// TwinCAT 3 PLC project Tc3_1CNCPLCBase
// Title: CNC PLC Project
// Company: Beckhoff Automation GmbH & Co. KG
// ProjectVersion: 3.1.3035.30
// ProgramVersion: 3.1.4020.0
// libraries:
//   Tc2_CncHli, * (Beckhoff Automation GmbH)
//   Tc2_Drive, * (Beckhoff Automation GmbH)
//   Tc2_EtherCAT, * (Beckhoff Automation GmbH)
//   Tc2_IoFunctions, * (Beckhoff Automation GmbH)
//   Tc2_Standard, * (Beckhoff Automation GmbH)
//   Tc2_System, * (Beckhoff Automation GmbH)
//   Tc2_Utilities, * (Beckhoff Automation GmbH)
//   Tc3_Module, * (Beckhoff Automation GmbH)
// project tree:
//   CNC Beckhoff/1 Init/ HLI3_InitToolConfig.TcPOU, HLI3_Init.TcPOU, HLI3_SetAxisControlToPlc.TcPOU, HLI3_SetChannelControlToPlc.TcPOU, HLI3_UserInitialisation.TcPOU
//   CNC Beckhoff/2 OperationMode/ HLI3_AxisReset.TcPOU, HLI3_ChannelModeAuto.TcPOU, HLI3_ChannelModeManual.TcPOU, HLI3_ChannelModeMDI.TcPOU, HLI3_ChannelModeReference.TcPOU, HLI3_ChannelModeStandby.TcPOU, HLI3_ChannelReset.TcPOU, HLI3_ChannelResetRequest.TcPOU, HLI3_CNCChannel.TcPOU
//   CNC Beckhoff/2 OperationMode/ModeManual/ HLI3_LogicalAxisInManualMode.TcPOU, HLI3_ManualActivation.TcPOU, HLI3_ManualExecution.TcPOU, HLI3_ManualExecutionRapidMode.TcPOU, HLI3_ManualModeHandler.TcPOU, PRG_AnalogJoystick.TcPOU
//   CNC Beckhoff/3 Control/ FB_Diag.TcPOU, HLI3_ChannelSetBackwardMotion.TcPOU, HLI3_ChannelSetEmergencyStop.TcPOU, HLI3_ChannelSetFeedHold.TcPOU, HLI3_ChannelSetProgramBlockIgnore.TcPOU, HLI3_ChannelSetReducedFeed.TcPOU, HLI3_ChannelSetSingleBlock.TcPOU, HLI3_ChannelSetSuspendAxisOutput.TcPOU, HLI3_ClearReferencePosition.TcPOU, HLI3_GetActualAxisPos.TcPOU, HLI3_GetAxisReferenceState.TcPOU, HLI3_GetChannelActiveG.TcPOU, HLI3_GetChannelError.TcPOU, HLI3_GetChannelMessage.TcPOU, HLI3_GetChannelMode.TcPOU, HLI3_GetChannelState.TcPOU, HLI3_GetChannelStatusInfo.TcPOU, HLI3_GetEtherCATAxisInfo.TcPOU, HLI3_GetFeedholdState.TcPOU, HLI3_GetIpoState.TcPOU, HLI3_HandleSpindleTechno.TcPOU, HLI3_HandleSpindleTechnoGearchange.TcPOU, HLI3_SetAxisGantryOn.TcPOU, HLI3_SetAxisOverride.TcPOU, HLI3_SetAxisReferenceCam.TcPOU, HLI3_SetAxisReferencePosition.TcPOU, HLI3_SetAxisRelease.TcPOU, HLI3_SetAxisSpindleStopAtProgramEnd.TcPOU, HLI3_SetAxisTrackingOperation.TcPOU, HLI3_SetChannelOverride.TcPOU, HLI3_SetProbingSignal.TcPOU
//   CNC Beckhoff/4 MHT-Function/ HLI3_ChannelResetHFunctions.TcPOU, HLI3_ChannelResetMFunctions.TcPOU, HLI3_DoChannelHFunction.TcPOU, HLI3_DoChannelMFunction.TcPOU, HLI3_DoChannelTFunction.TcPOU, HLI3_FastMFunctionHandler.TcPOU, HLI3_FastMFunctionProvider.TcPOU, HLI3_QuitAxisMFunction.TcPOU, HLI3_QuitChannelMHTFunction.TcPOU, PRG_FastMFunctions.TcPOU
//   CNC Beckhoff/5 Variables/ FB_ReadCNCVariables.TcPOU, HLI3_GetVEChannelDIntValue.TcPOU, HLI3_GetVEChannelBooleanValue.TcPOU, HLI3_GetVEChannelLRealValue.TcPOU, HLI3_GetVEChannelStringValue.TcPOU, HLI3_LinkVEChannelStructure.TcPOU, HLI3_SetVEChannelDIntValue.TcPOU, HLI3_SetVEChannelBooleanValue.TcPOU, HLI3_SetVEChannelLRealValue.TcPOU, HLI3_SetVEChannelStringValue.TcPOU
//   CNC Beckhoff/6 BlockSearch/ HLI3_BlockSearch.TcPOU, ReadBlockCount.TcPOU, ReadBlockNumber.TcPOU, ReadBsAutoReturn.TcPOU, ReadBsBlockCount.TcPOU, ReadBsBlockNumber.TcPOU, ReadBsCoveredDistance.TcPOU, ReadBsDeviationMax.TcPOU, ReadBsPass.TcPOU, ReadBsType.TcPOU, WriteBsAutoReturn.TcPOU, WriteBsBlockCount.TcPOU, WriteBsBlockNumber.TcPOU, WriteBsCoveredDistance.TcPOU, WriteBsDeviationMax.TcPOU, WriteBsPass.TcPOU, WriteBsType.TcPOU
//   CNC Beckhoff/9 Mis/ ADSLOG.TcPOU, FB_WriteCNCZeroOffset.TcPOU, FB_WriteCNCZeroOffsetDefault.TcPOU, HLI3_CheckAxisValid.TcPOU, HLI3_CheckChannelValid.TcPOU, HLI3_CheckCNCAlive.TcPOU, HLI3_GetHliAxisIdx.TcPOU, HLI3_GetLogAxisId.TcPOU, HLI3_SetPLCAlive.TcPOU, HLI_HandleMessages.TcPOU, HLI_MoveSpindle.TcPOU, PB_10_CNC_Spindelkopplung.TcPOU, HLI3_ResetSpindle.TcPOU
//   CNC Beckhoff/Demo/ PRG_Demo.TcPOU, PRG_MachineStatusV2.TcPOU
//   CNC Beckhoff/Messages/ FB_ChannelError.TcPOU, FB_EventLog.TcPOU, FB_ExtSimpleEventLog.TcPOU, FB_SimpleEventLog.TcPOU
//   CNC Beckhoff/ PRG_AxesHandler.TcPOU, PRG_ChannelHandler.TcPOU, PRG_CNCVariablesViewer.TcPOU, PRG_ManualMode.TcPOU, PRG_ManualModeHMI.TcPOU, PRG_ShowMessages.TcPOU
//   CNC Beckhoff/Util/ Blinker.TcPOU, FB_CNCWriteParameter.TcPOU, FB_Uint_Udint.TcPOU, F_GRAYCODE_TO_UINT.TcPOU, HLI3_FindHliAxisIdx.TcPOU, HLI3_FindAxisNameAndChannel.TcPOU
//   Data types/CNC_DataTyps/ E_CNC_MM_Controller.TcDUT, E_HLI_MM_KEYDIRECTION.TcDUT, ST_BlockSearch.TcDUT, ST_ChannelSignals.TcDUT, ST_CNCAxis.TcDUT, ST_CncChannel.TcDUT, ST_CNCG159VG.TcDUT, ST_CncSystem.TcDUT, ST_CNC_TOOL_DATA_EXT.TcDUT, ST_ManualMode.TcDUT, ST_OpModes.TcDUT, ST_OpStates.TcDUT, ST_SyntaxCheck.TcDUT, ST_TechnoAttributeData.TcDUT, VEData.TcDUT
//   Data types/CNC_FastMFunction/ E_FastMFunctionState.TcDUT, ST_FastMFunctionBufferItem.TcDUT, ST_FastMFunctionData.TcDUT, ST_FastMFunctionItem.TcDUT
//   Data types/CNC_ManualMode/ E_CNC_ManualType.TcDUT, ST_ManualModeAxis.TcDUT, ST_ManualModeAxisKeys.TcDUT, ST_ManualModeAxisParameter.TcDUT, ST_ManualModeChannelParameter.TcDUT, ST_ManualModeControlElements.TcDUT, ST_ManualModeControlElementState.TcDUT, ST_ManualModeJoystickParameter.TcDUT, ST_ManualModeKeyHWUnit.TcDUT, ST_ManualModeParameter.TcDUT, ST_ManualModeState.TcDUT
//   Data types/CNC_VariablesViewer/ E_CNCVariablesType.TcDUT, E_VEVariablesType.TcDUT, ST_CNCVariablesViewer_Data.TcDUT
//   Data types/CNC_WriteParameter/ E_CNCParameterTypes.TcDUT, ST_CNCParameter.TcDUT
//   Data types/EtherCAT Diag/ E_EcCommState.TcDUT, ST_EcMasterDevState.TcDUT, ST_PortAddr.TcDUT, ST_SlaveState.TcDUT, ST_SlaveStateInfo.TcDUT, ST_SlaveStateInfoScanned.TcDUT, ST_TopologyData.TcDUT
//   Data types/EventLogger/ E_LogMethod.TcDUT, ST_EventData.TcDUT, ST_FileInfo.TcDUT
//   Data types/ E_HLI_MM_STATE.TcDUT, ST_Diagnose.TcDUT, ST_EtherCATAxisInfo.TcDUT, ST_EventData1.TcDUT, ST_EventDataAX5000_1.TcDUT, ST_MachineMode.TcDUT, ST_MViewStatus.TcDUT, ST_WKZDaten.TcDUT, ST_WPCounter.TcDUT
//   Data types/General SoE DTs/ ST_SoE_String.TcDUT, ST_SoE_StringEx.TcDUT
//   Data types/Magazin/ ST_Magazin.TcDUT
//   Data types/MaschinenDaten PlcStructure/ ST_HMIPDatMaschine.TcDUT, ST_HMIPDatProg.TcDUT, ST_HMI_Manual.TcDUT, ST_MachData.TcDUT, ST_PDatLineProgLine.TcDUT, ST_PDatLineProgValue.TcDUT
//   Data types/Recipe/ RecipeHeader_Struct.TcDUT, RecipeList_Struct.TcDUT
//   Data types/SERCOS/ E_SoE_AttribLen.TcDUT, E_SoE_CmdControl.TcDUT, E_SoE_CmdState.TcDUT, E_SoE_Type.TcDUT
//   / FAST.TcPOU, MAIN.TcPOU, PlcFastTask.TcTTO, Standard_Task.TcTTO
//   Global Variables/Examples/ Globale_EtherCATDiag.TcGVL, Global_BDE.TcGVL, Global_MachineView.TcGVL, Global_ManualPlcFunctions.TcGVL, Global_MaschinenDaten.TcGVL, Global_VE.TcGVL
//   Global Variables/ Global_CNC.TcGVL, Global_CNCVariablesViewer.TcGVL, Global_HMI.TcGVL, Global_ManualMode.TcGVL, Global_Messages.TcGVL, Variable_Configuration.TcGVL
//   Version/ Global_Version.TcGVL
// real-time tasks:
//   TASK Standard_Task: cycle T#10ms, priority 21, ADS port 350
//   TASK PlcFastTask: cycle T#1ms, priority 4, ADS port 351
// I/O:
//   DEVICE Gerät 3 (EtherCAT), AmsNetId 10.99.10.27.4.1
//     testachse [AX5103-0000-0203 EtherCAT Drive (SoE, 1 Ch.)] (disabled)
//     Drive 2 (AX5206-0000-0011) [AX5206-0000 EtherCAT Drive (SoE, 2 Ch.)]
// variable links:
//   CNC/Axes/Axis_2 <-> Device 3 (EtherCAT)/Drive 2 (AX5206-0000-0011)
//     Inputs/Drive status word <-> AT 1/Drive status word
//     Inputs/Following distance <-> AT 1/Following distance
//     Inputs/Position feedback value 1 (motor feedback) <-> AT 1/Position feedback value 1 (motor feedback)
//     Inputs/WcState <-> WcState/WcState
//     Outputs/Master control word <-> MDT 1/Master control word
//     Outputs/Position command value <-> MDT 1/Position command value
//   CNC/Axes/Axis_3 <-> Device 3 (EtherCAT)/Drive 2 (AX5206-0000-0011)
//     Inputs/Drive status word <-> AT 2/Drive status word
//     Inputs/Following distance <-> AT 2/Following distance
//     Inputs/Position feedback value 1 (motor feedback) <-> AT 2/Position feedback value 1 (motor feedback)
//     Inputs/WcState <-> WcState/WcState
//     Outputs/Master control word <-> MDT 2/Master control word
//     Outputs/Position command value <-> MDT 2/Position command value
//   Tc3_1CNCPLCBase/Tc3_1CNCPLCBase Instance <-> Device 3 (EtherCAT)/Drive 2 (AX5206-0000-0011)
//     Standard_Task Inputs/MAIN.DigitalIn <-> AT 1/Digital inputs, state
//     Standard_Task Outputs/MAIN.Trennscheibe <-> MDT 1/Digital outputs

CONFIGURATION Tc3_1CNCPLCBase
    RESOURCE PLC ON TwinCAT3
        TASK PlcFastTask(INTERVAL := T#1ms, PRIORITY := 4);
        TASK Standard_Task(INTERVAL := T#10ms, PRIORITY := 21);
        PROGRAM FAST WITH PlcFastTask : FAST;
        PROGRAM MAIN WITH Standard_Task : MAIN;
    END_RESOURCE
END_CONFIGURATION

// ---- Data types/CNC_DataTyps/E_CNC_MM_Controller.TcDUT
TYPE E_CNC_MM_Controller :
(
	HMI := 0,
	PANEL := 1,
	REMOTE := 2,
	CUSTOMER := 3
);
END_TYPE

// ---- Data types/CNC_DataTyps/E_HLI_MM_KEYDIRECTION.TcDUT
TYPE E_HLI_MM_KEYDIRECTION :
(
	KEY_DIR_NEGATIVE := -1,
	KEY_DIR_NOT_PRESSED := 0,
	KEY_DIR_POSITIVE := 1
);
END_TYPE

// ---- Data types/CNC_DataTyps/ST_BlockSearch.TcDUT
TYPE ST_BlockSearch :
STRUCT
	/// Block Search 
	Active: BOOL;
	/// Edge signal 
	bStartRead: BOOL;
	/// Edge signal 
	bStartWrite: BOOL;
	/// 0 - no block search
	///                                    3 - start position by block count
	///                                    4 - start position by block nr
	///                                    5 - start position BY individual mark 
	nType: UINT;
	fDistance: LREAL;
	bAutoReturn: BOOL;
	nDeviationMax: UDINT;
	nBlockNumber: DINT;
	nPass: DINT;
	nBlockCount: DINT;
END_STRUCT
END_TYPE

// ---- Data types/CNC_DataTyps/ST_ChannelSignals.TcDUT
TYPE ST_ChannelSignals :
STRUCT
	DoSingleBlock: BOOL;
	SingleBlock: BOOL;
	FeedHold: BOOL;
	Backward: BOOL;
	PrgBlockIgnore: BOOL;
	M01Stop: BOOL;
END_STRUCT
END_TYPE

// ---- Data types/CNC_DataTyps/ST_CNCAxis.TcDUT
TYPE ST_CNCAxis :
STRUCT
	nHliAxisIdx : INT := -1;
    stLogName	: STRING(HLI_ACHS_NAME_LAENGE);
END_STRUCT
END_TYPE

// ---- Data types/CNC_DataTyps/ST_CncChannel.TcDUT
TYPE ST_CncChannel :
STRUCT
	/// Operation Mode 
	Mode: ST_OpModes;
	/// Operation States 
	State: ST_OpStates;
	/// Selected Mode 
	ActMode: UDINT;
	/// Selected Mode as string 
	ActModeString: STRING;
	/// Selected State 
	ActState: UDINT;
	/// Selected State as string 
	ActStateString: STRING;
	/// Block Search : Act. Distance 
	ActDistance: LREAL;
	/// Block Search : Act. Block Count 
	ActBlockCount: UDINT;
	actM_r: STRING(5);
	actH_r: STRING(5);
	/// M-Functions 
	M: ARRAY[0..999] OF ST_TechnoAttributeData;
	/// H-Functions 
	H: ARRAY[0..999] OF ST_TechnoAttributeData;	
	/// Fehlerflag des Kanals 
	Error: BOOL;	
	/// Message from NC program to PLC 
	Message: STRING(HLI_MSG_CONTENT_STRL);
END_STRUCT
END_TYPE

// ---- Data types/CNC_DataTyps/ST_CNCG159VG.TcDUT
TYPE ST_CNCG159VG :
STRUCT
	sTarget: STRING(95);
	dValue: DINT;
END_STRUCT
END_TYPE

// ---- Data types/CNC_DataTyps/ST_CncSystem.TcDUT
TYPE ST_CncSystem :
STRUCT
	/// Initialization of HLI done 
	bHLIInit: BOOL;
	/// Initialization of user data done 
	bUserInitDone: BOOL;
	/// Error init HLI-Interfaces 
	bInitError: BOOL;
	/// ErrorId during init HLI-Interfaces 
	nInitErrorId: UDINT;
	Channel: ARRAY[0..HLI_SYS_CH_MAXIDX] OF ST_CncChannel;
    LogAxisNo : ARRAY[0..MAX_SYS_LOG_AXIS_INDEX] OF ST_CncAxis;	
END_STRUCT
END_TYPE

// ---- Data types/CNC_DataTyps/ST_CNC_TOOL_DATA_EXT.TcDUT
TYPE ST_CNC_TOOL_DATA_EXT :
STRUCT
	tool_desc: CNC_TOOL_DESC;
	tool_life: CNC_TOOL_LIFE_DATA;
	dist_max: LREAL;
	time_max: LREAL;
	/// 0.1 µm 
	laenge: DINT;
	/// 0.1 µm 
	laenge_delta: DINT;
	/// 0.1 µm 
	radius: DINT;
	/// 0.1 µm 
	radius_delta: DINT;
	/// position in tool holder 
	pos: DINT;
	/// 0.1 µm 
	tolerancePos: DINT;
	/// 0.1 µm 
	toleranceNeg: DINT;
END_STRUCT
END_TYPE

// ---- Data types/CNC_DataTyps/ST_ManualMode.TcDUT
TYPE ST_ManualMode :
STRUCT
	bKeyPos: BOOL;
	bKeyNeg: BOOL;
	bKeyRapid: BOOL;
	nLogAxisNumber: UINT;
	nInc: UDINT;
	nManualTyp: UINT;
	nSpeed: UINT;
	/// Handradauflösung in 0.1 um / Umdrehung 
	nHwResolution: UDINT;
END_STRUCT
END_TYPE

// ---- Data types/CNC_DataTyps/ST_OpModes.TcDUT
TYPE ST_OpModes :
STRUCT
	Standby: BOOL;
	Auto: BOOL;
	Manual: BOOL;
	MDI: BOOL;
	///Reference		: BOOL;  TC3HR
	Homing: BOOL;
END_STRUCT
END_TYPE

// ---- Data types/CNC_DataTyps/ST_OpStates.TcDUT
TYPE ST_OpStates :
STRUCT
	Selected: BOOL;
	Ready: BOOL;
	Start: BOOL;
	Stop: BOOL;
	Reset: BOOL;
END_STRUCT
END_TYPE

// ---- Data types/CNC_DataTyps/ST_SyntaxCheck.TcDUT
TYPE ST_SyntaxCheck :
STRUCT
	/// SyntaxCheck 
	nType: INT;
END_STRUCT
END_TYPE

// ---- Data types/CNC_DataTyps/ST_TechnoAttributeData.TcDUT
TYPE ST_TechnoAttributeData :
STRUCT
	bState_rw: BOOL;
	nFunctionNumber_r: UDINT;
	nTime_r: DINT;
	nBlockNumber_r: UDINT;
	nPrgLineNumber_r: UDINT;
	nArgument_r: DINT;
	bRes: BOOL;
END_STRUCT
END_TYPE

// ---- Data types/CNC_DataTyps/VEData.TcDUT
TYPE VEData :
STRUCT
	AHLI_UNS32_Data: ARRAY[0..HLI_EXT_VAR32_MAXIDX] OF UDINT;
END_STRUCT
END_TYPE

// ---- Data types/CNC_FastMFunction/E_FastMFunctionState.TcDUT
(****************************************************************************************)
(* POU:		E_FastMFunctionState                     									*)
(* Type:	ENUM																		*)
(* Author: 	RCH		                                             						*)
(* Date: 	14/10/29																	*)
(* Rev.: 	1.0                                               							*)
(* ------------------------------------------------------------------------------------ *)
(* Desc.:	Defines the state of an digital output handled by instances of FB			*)
(*			HLI3_FastMFunctionHandler.													*)
(* ------------------------------------------------------------------------------------ *)
(* Rev.:	<Enter revision number here>												*)
(* Date:	<Enter revision data here>				                                   	*)
(* Author:	<Enter author´s shortcut here>											 	*)
(* Desc.:	<Enter description here>													*)
(****************************************************************************************)
TYPE E_FastMFunctionState :
(
	EMPTY	:= 0,	(* Not switched yet *)
	OFF 	:= 1,	(* Switched OFF *)
	ON 		:= 2	(* Switched ON *)
);
END_TYPE

// ---- Data types/CNC_FastMFunction/ST_FastMFunctionBufferItem.TcDUT
(****************************************************************************************)
(* POU:		ST_FastMFunctionBufferItem                     								*)
(* Type:	STRUCT																		*)
(* Author: 	RCH		                                             						*)
(* Date: 	14/10/29																	*)
(* Rev.: 	1.0                                               							*)
(* ------------------------------------------------------------------------------------ *)
(* Desc.:	Defines data content for a single fast M function switch event managed 		*)
(*			internally by instances of HLI3_FastMFunctionHandler.						*) 
(* ------------------------------------------------------------------------------------ *)
(* Rev.:	<Enter revision number here>												*)
(* Date:	<Enter revision data here>				                                   	*)
(* Author:	<Enter author´s shortcut here>											 	*)
(* Desc.:	<Enter description here>													*)
(****************************************************************************************)
TYPE ST_FastMFunctionBufferItem :
STRUCT
	eState			: E_FastMFunctionState;		(* The target switch state *)
	nSwitchTime		: DINT;						(* The calculated switch time *)
END_STRUCT
END_TYPE

// ---- Data types/CNC_FastMFunction/ST_FastMFunctionData.TcDUT
(****************************************************************************************)
(* POU:		ST_FastMFunctionData                     								*)
(* Type:	STRUCT																		*)
(* Author: 	RCH		                                             						*)
(* Date: 	14/10/29																	*)
(* Rev.: 	1.0                                               							*)
(* ------------------------------------------------------------------------------------ *)
(* Desc.:	Defines preprocessed information about MOS_TS M functions and their			*)
(*			metadata generated by HLI3_FastMFunctionProvider and consumed by 			*)
(*			HLI3_FastMFunctionHandler(s)												*) 
(* ------------------------------------------------------------------------------------ *)
(* Rev.:	<Enter revision number here>												*)
(* Date:	<Enter revision data here>				                                   	*)
(* Author:	<Enter author´s shortcut here>											 	*)
(* Desc.:	<Enter description here>													*)
(****************************************************************************************)
TYPE ST_FastMFunctionData :
STRUCT
	bCycleTimeExceeded	: BOOL;																	(* TRUE if the cycle time has been exceeded and therefore the data is unvalid *)
	bDataValid			: BOOL;																	(* TRUE if data is valid *)
	nFunctionCount		: UINT;																	(* Number of M function data sets contained in 'astItem' *)
	astItem				: ARRAY[0..MAX_FAST_M_FUNC_ITEM_IDX] OF ST_FastMFunctionItem;			(* M function metadata items *)
END_STRUCT
END_TYPE

// ---- Data types/CNC_FastMFunction/ST_FastMFunctionItem.TcDUT
(****************************************************************************************)
(* POU:		ST_FastMFunctionItem                     									*)
(* Type:	STRUCT																		*)
(* Author: 	RCH		                                             						*)
(* Date: 	14/10/29																	*)
(* Rev.: 	1.0                                               							*)
(* ------------------------------------------------------------------------------------ *)
(* Desc.:	Defines M function metadata content provided by HLI3_FastMFunctionProvider	*)
(* ------------------------------------------------------------------------------------ *)
(* Rev.:	<Enter revision number here>												*)
(* Date:	<Enter revision data here>				                                   	*)
(* Author:	<Enter author´s shortcut here>											 	*)
(* Desc.:	<Enter description here>													*)
(****************************************************************************************)
TYPE ST_FastMFunctionItem :
STRUCT
	nFunctionNo		: UINT;			(* M function number *)
	nOffset			: DINT;			(* Time offset with respect to the block change time *)
	nCycleCount		: UDINT;		(* PLC cycle counter *)
END_STRUCT
END_TYPE

// ---- Data types/CNC_ManualMode/E_CNC_ManualType.TcDUT
TYPE E_CNC_ManualType :
(
	NoManualMode := 0,
	Handwheel := 1,
	TippMode := 2,
	JogMode := 3,
	JoystickMode := 4,
	DigitalJoystick := 5
);
END_TYPE

// ---- Data types/CNC_ManualMode/ST_ManualModeAxis.TcDUT
TYPE ST_ManualModeAxis :
STRUCT
	nLogAxisNr: UINT;
	nSpeed: UDINT;
END_STRUCT
END_TYPE

// ---- Data types/CNC_ManualMode/ST_ManualModeAxisKeys.TcDUT
TYPE ST_ManualModeAxisKeys :
STRUCT
	/// static signal + 
	bKeyPos: BOOL;
	/// static signal - 
	bKeyNeg: BOOL;
	/// static signal Rapid 
	bKeyRapid: BOOL;
END_STRUCT
END_TYPE

// ---- Data types/CNC_ManualMode/ST_ManualModeAxisParameter.TcDUT
TYPE ST_ManualModeAxisParameter :
STRUCT
	stControlUnit: ARRAY[0..HLI_KEY_MAXIDX] OF ST_ManualModeAxis;
END_STRUCT
END_TYPE

// ---- Data types/CNC_ManualMode/ST_ManualModeChannelParameter.TcDUT
TYPE ST_ManualModeChannelParameter :
STRUCT
	/// Number of channel 
	nChanIdx: INT := -1;
	nInc: UDINT;
	/// Aufloesung des Achsverfahrwegs bei einer Handradumdrehung Einheit: 0.1um / Handradumdrehung
	nHandwheelResolution: DINT;	 	
	/// configuration 
	eManualType: E_CNC_ManualType;
	strInitParameter: STRING;
END_STRUCT
END_TYPE

// ---- Data types/CNC_ManualMode/ST_ManualModeControlElements.TcDUT
TYPE ST_ManualModeControlElements :
STRUCT
	stControlKeys: ARRAY[0..HLI_KEY_MAXIDX] OF ST_ManualModeAxisKeys;
	stControlJoystickValue: ARRAY[0..HLI_KEY_MAXIDX] OF DINT;
	/// Es können 6 Handräder verwendet werden 
	nHandwheelInc: ARRAY[0..HLI_HW_MAXIDX] OF DINT;
END_STRUCT
END_TYPE

// ---- Data types/CNC_ManualMode/ST_ManualModeControlElementState.TcDUT
TYPE ST_ManualModeControlElementState :
STRUCT
	stKeyUnit: ARRAY[0..HLI_KEY_MAXIDX] OF ST_ManualModeKeyHWUnit;
	stHWUnit: ARRAY[0..HLI_HW_MAXIDX] OF ST_ManualModeKeyHWUnit;
END_STRUCT
END_TYPE

// ---- Data types/CNC_ManualMode/ST_ManualModeJoystickParameter.TcDUT
TYPE ST_ManualModeJoystickParameter :
STRUCT
	/// static signal : Analog Min Value 
	AnalogValueMin: DINT;
	/// static signal : Analog Max Value 
	AnalogValueMax: DINT;
	/// Dead Band for Zero Value 
	AnalogValueZeroDeadBand: DINT;
END_STRUCT
END_TYPE

// ---- Data types/CNC_ManualMode/ST_ManualModeKeyHWUnit.TcDUT
TYPE ST_ManualModeKeyHWUnit :
STRUCT
	nLogAxisId: UINT;
	nChan: INT := -1;
	nInputParameterIdx: INT;
END_STRUCT
END_TYPE

// ---- Data types/CNC_ManualMode/ST_ManualModeParameter.TcDUT
TYPE ST_ManualModeParameter :
STRUCT
	stAxisParameter: ST_ManualModeAxisParameter;
	stJoystickParameter: ST_ManualModeJoystickParameter;
	stChannelParameter: ST_ManualModeChannelParameter;	
END_STRUCT
END_TYPE

// ---- Data types/CNC_ManualMode/ST_ManualModeState.TcDUT
TYPE ST_ManualModeState :
STRUCT
	arrAxisInG201: ARRAY[0..HLI_KEY_MAXIDX] OF UINT;
END_STRUCT
END_TYPE

// ---- Data types/CNC_VariablesViewer/E_CNCVariablesType.TcDUT
{attribute 'qualified_only'}
{attribute 'strict'}
TYPE E_CNCVariablesType :
(
	none :=0,
	VE,
    P,
    VP,
    VS,
    VL,
    VG,
    VA
);
END_TYPE

// ---- Data types/CNC_VariablesViewer/E_VEVariablesType.TcDUT
{attribute 'qualified_only'}
{attribute 'strict'}
TYPE E_VEVariablesType :
(
	none := 0,
	BOOLEAN,
	SGN08,
	UNS08,
	SGN16,
	UNS16,
	SGN32,
	UNS32,
	REAL64,
	VESTRING
);
END_TYPE

// ---- Data types/CNC_VariablesViewer/ST_CNCVariablesViewer_Data.TcDUT
TYPE ST_CNCVariablesViewer_Data :
STRUCT
	strName : STRING;
	strValue  : STRING(127);
END_STRUCT
END_TYPE

// ---- Data types/CNC_WriteParameter/E_CNCParameterTypes.TcDUT
TYPE E_CNCParameterTypes :
(
	CNC_ChannelParameter := 10,
	CNC_AxisParameter := 11,
	CNC_ZeroOffsets := 12,
	CNC_ToolParameter := 13,
	CNC_ClampPosition := 14
);
END_TYPE

// ---- Data types/CNC_WriteParameter/ST_CNCParameter.TcDUT
TYPE ST_CNCParameter :
STRUCT
	strName: STRING;
	strValue: STRING;
	strDescription: STRING;
END_STRUCT
END_TYPE

// ---- Data types/EtherCAT Diag/E_EcCommState.TcDUT
TYPE E_EcCommState :
(
	eEcState_UNDEFINED := 0,
	eEcState_INIT := 1,
	eEcState_PREOP := 2,
	eEcState_BOOT := 3,
	eEcState_SAFEOP := 4,
	eEcState_OP := 8
);
END_TYPE

// ---- Data types/EtherCAT Diag/ST_EcMasterDevState.TcDUT
TYPE ST_EcMasterDevState :
STRUCT
	eEcState: E_EcCommState;
	nReserved: ARRAY[0..2] OF UINT;
	bLinkError: BOOL;
	bResetRequired: BOOL;
	bMissFrmRedMode: BOOL;
	bWatchdogTriggerd: BOOL;
	bDriverNotFound: BOOL;
	bResetActive: BOOL;
	bAtLeastOneNotInOp: BOOL;
	bDcNotInSync: BOOL;
END_STRUCT
END_TYPE

// ---- Data types/EtherCAT Diag/ST_PortAddr.TcDUT
TYPE ST_PortAddr :
STRUCT
	portA: UINT;
	portB: UINT;
	portC: UINT;
	portD: UINT;
END_STRUCT
END_TYPE

// ---- Data types/EtherCAT Diag/ST_SlaveState.TcDUT
TYPE ST_SlaveState :
STRUCT
	/// slave state 
	eEcState: E_EcCommState;
	nReserved: UINT;
	bError: BOOL;
	bInvalidVPRS: BOOL;
	nReserved2: UINT;
	/// link state 
	bNoCommToSlave: BOOL;
	bLinkError: BOOL;
	bMissingLink: BOOL;
	bUnexpectedLink: BOOL;
	bPortA: BOOL;
	bPortB: BOOL;
	bPortC: BOOL;
	bPortD: BOOL;
END_STRUCT
END_TYPE

// ---- Data types/EtherCAT Diag/ST_SlaveStateInfo.TcDUT
TYPE ST_SlaveStateInfo :
STRUCT
	nIndex: DINT;
	/// name of slave given in System Manager 
	sName: STRING;
	/// type of slave, e.g. EK1100
	sType: STRING;
	/// EtherCAT Slave Addr 
	nECAddr: UINT;
	/// DiagData in Slave State 
	bDiagData: BOOL;
	/// Slave CRC-Errors, separate for each Port 
	stPortCRCErrors: ST_EcCrcErrorEx;
	/// Slave CRC-Errors, sum of all Ports 
	nSumCRCErrors: UDINT;
	/// EtherCAT State and Link state
	stState: ST_SlaveState;
END_STRUCT
END_TYPE

// ---- Data types/EtherCAT Diag/ST_SlaveStateInfoScanned.TcDUT
TYPE ST_SlaveStateInfoScanned :
STRUCT
	nIndex: DINT;
	/// name of slave given in System Manager 
	sName: STRING;
	/// type of slave, e.g. EK1100
	sType: STRING;
	/// EtherCAT Slave Addr 
	nECAddr: UINT;
	/// Name of Scanned configuration differs from Configured configuration 
	bDifferentName: BOOL;
	/// Type Of Scanned configuration differs from Configured configuration 
	bDifferentType: BOOL;
	/// EcAddress of Scanned configuration differs from Configured configuration 
	bDifferentAddr: BOOL;
END_STRUCT
END_TYPE

// ---- Data types/EtherCAT Diag/ST_TopologyData.TcDUT
TYPE ST_TopologyData :
STRUCT
	iOwnPhysicalAddr: UINT;
	iOwnAutoIncAddr: UINT;
	stPhysicalAddr: ST_PortAddr;
	stAutoIncAddr: ST_PortAddr;
	/// EC_AD, EC_DB, EC_BC 
	iPortDelay: ARRAY[0..2] OF UDINT;
	iReserved: ARRAY[0..7] OF UDINT;
END_STRUCT
END_TYPE

// ---- Data types/EventLogger/E_LogMethod.TcDUT
TYPE E_LogMethod :
(
	Static := 0,
	RisingTrig := 1,
	FallingTrig := 2
);
END_TYPE

// ---- Data types/EventLogger/ST_EventData.TcDUT
TYPE ST_EventData :
STRUCT
	nSourceText: UINT;
	nSourceDesc: UINT;
	nErrorCode: UDINT;
	sModul: STRING;
	sAddInfo: STRING;
END_STRUCT
END_TYPE

// ---- Data types/EventLogger/ST_FileInfo.TcDUT
TYPE ST_FileInfo :
STRUCT
	nSource: UDINT;
	nOffset: UDINT;
	sFilename: STRING(260);
END_STRUCT
END_TYPE

// ---- Data types/E_HLI_MM_STATE.TcDUT
TYPE E_HLI_MM_STATE :
(
	SMM_ERROR := -1,
	/// axis to the 2.channel                     
	SMM_SUSPEND_AXIS_CHAN1 := 0,
	/// wait for suspension of the 1.channel      
	SMM_SUSPEND_AXIS_CHAN1_WAIT,
	SMM_STORE_POSITION,
	SMM_INIT_MANUAL_MODE,
	SMM_SWITCH_TO_M_READY,
	SMM_SWITCH_TO_M_READY_WAIT,
	SMM_STATUS_READY,
	/// wait for direction input                  
	SMM_WAIT_FOR_ACTIVATE,
	/// switch to manual-mode                     
	SMM_SWITCH_TO_M_MODE,
	/// wait for manual-mode switch               
	SMM_SWITCH_TO_M_MODE_WAIT,
	/// parametrize, tip parameter                
	SMM_SET_TIP_PARAM_AXIS1,
	/// wait for parametrize, tip parameter       
	SMM_SET_TIP_PARAM_AXIS1_WAIT,
	/// parametrize, tip parameter                
	SMM_SET_TIP_PARAM_AXIS2,
	/// wait for parametrize, tip parameter       
	SMM_SET_TIP_PARAM_AXIS2_WAIT,
	/// activate tip mode axis 1                  
	SMM_ACTIVE_TIP_MODE_AXIS1,
	/// wait for parametrize, tip mode axis 1     
	SMM_ACTIVE_TIP_MODE_AXIS1_WAIT,
	/// activate tip mode axis 2                  
	SMM_ACTIVE_TIP_MODE_AXIS2,
	/// wait for parametrize, tip mode axis 2     
	SMM_ACTIVE_TIP_MODE_AXIS2_WAIT,
	/// control manual mode axis 1 and axis 2     
	SMM_CONTROL_M_MODE,
	/// deactivate tip mode axis 1                
	SMM_DEACTIVE_TIP_MODE_AXIS1,
	/// wait for deactivating, tip mode axis 1    
	SMM_DEACTIVE_TIP_MODE_AXIS1_WAIT,
	/// deactivate tip mode axis 2                
	SMM_DEACTIVE_TIP_MODE_AXIS2,
	/// wait for deactivating, tip mode axis 2    
	SMM_DEACTIVE_TIP_MODE_AXIS2_WAIT,
	/// move back or end                          
	SMM_MOVEBACK_OR_END,
	/// MDI mode switch and activation            
	SMM_ACTIVATE_MDI_MODE,
	/// wait for MDI mode switch and activation   
	SMM_ACTIVATE_MDI_MODE_WAIT,
	/// wait for MDI movement                     
	SMM_PROCESS_READY_MDI_MODE,
	/// axis to the 1.channel                     
	SMM_SUSPEND_AXIS_CHAN2
);
END_TYPE

// ---- Data types/General SoE DTs/ST_SoE_String.TcDUT
TYPE ST_SoE_String :
STRUCT
	iActualSize: UINT;
	iMaxSize: UINT;
	strData: STRING(MAX_STRING_LENGTH);
END_STRUCT
END_TYPE

// ---- Data types/General SoE DTs/ST_SoE_StringEx.TcDUT
TYPE ST_SoE_StringEx :
STRUCT
	dwAttribute: DWORD;
	iActualSize: UINT;
	iMaxSize: UINT;
	strData: STRING(MAX_STRING_LENGTH);
END_STRUCT
END_TYPE

// ---- Data types/Magazin/ST_Magazin.TcDUT
TYPE ST_Magazin :
STRUCT
	bPlatzBelegt: ARRAY[1..8] OF BOOL;
	id: ARRAY[1..8] OF CNC_TOOL_ID;
END_STRUCT
END_TYPE

// ---- Data types/MaschinenDaten PlcStructure/ST_HMIPDatMaschine.TcDUT
TYPE ST_HMIPDatMaschine :
STRUCT
	///@1: Überstand @11:2
	arrOverhang: ARRAY[1..2] OF LREAL;
	/// @1: Vorschubgeschwindigkeit @11:2
	fFeedVelo: LREAL;
	///@1:Filename @5:1 @11:2
	sFileName: STRING(255);
	/// @1: Kantenfarbe @11:2
	arrEdgecolor: ARRAY[1..2] OF DINT;
	/// @1: Unterprogramm @11:2
	arrProg: ARRAY[1..4] OF ST_HMIPDatProg;
END_STRUCT
END_TYPE

// ---- Data types/MaschinenDaten PlcStructure/ST_HMIPDatProg.TcDUT
TYPE ST_HMIPDatProg :
STRUCT
	/// @1: Bearbeitung @11:2
	nWorking: INT;
	/// @1: Streckenwerte @11:2
	stLine: ST_PDatLineProgLine;
	/// @1: Werte mit Verstellung @11:2
	stAdjustment: ST_PDatLineProgValue;
	/// @1: Werte ohne Verstellung @11:2
	stNoAdjustment: ST_PDatLineProgValue;
END_STRUCT
END_TYPE

// ---- Data types/MaschinenDaten PlcStructure/ST_HMI_Manual.TcDUT
TYPE ST_HMI_Manual :
STRUCT
	/// @1:Beschreibung @11:1 @2: 1.Spalte Beschreibung:0=tastend, 1 =rastend @3 2.Spalte Beschreibung:0=tastend, 1 =rastend ...
	/// Milling 
	milling: BYTE;
	millingStatus: BYTE;
	/// Blowing
	/// @1:abblasen @11:1 @2:on:1 @3:Position 1 Super @4:Position 2 auf Taste2 @5:Position 3 @6: Pos 4 @7: Disable @8:Pos8 @9: Position 9 
	blowing: BYTE;	
	blowingStatus: BYTE;
	/// Axis 
	axisY: BYTE;
	axisYStatus: BYTE;
	/// @1:Z-Axis @11:1 @2:Forward:0 @3:Backward:0
	axisZ: BYTE;
	axisZStatus: BYTE;
	/// @1:C-Axis @11:1 @2:Forward:0 @3:Backward:0
	axisC: BYTE;
	axisCStatus: BYTE;
	/// @1:U-Axis @11:1 @2:Forward:0 @3:Backward:0 @5:Grundpos
	axisU: BYTE;
	axisUStatus: BYTE;
	/// @1:V-Axis @11:1 @2:Forward:0 @3:Backward:0 @5:Grundpos
	axisV: BYTE;
	axisVStatus: BYTE;
	
END_STRUCT
END_TYPE

// ---- Data types/MaschinenDaten PlcStructure/ST_MachData.TcDUT
TYPE ST_MachData :
STRUCT
	/// @1:Aktivflag @11:2
	bAktiv: BOOL;
	///@1: Wert 1 @11:2
	nWert12: INT;
	///@1: Wert 2 @11:2
	nWert2: INT;
	///@1: Auftrags-ID @11:2
	nAuftragId: DINT;
	///@1:ProdHandle @11:2
	nProdHandle: DINT;
	///@1:Barcode @11:2
	sBarcode: STRING;
	///@1:Zeit
	Zeit: TIME;
	///Dateiname
	sFileName: STRING;
	///Sollstückzahl
	nSetPiece: DINT;
	///Iststückzahl
	nActPiece: DINT;
	///Name-Unterprogramm1
	sUProg1: STRING;
	///Name-Unterprogramm2
	sUProg2: STRING;
	///Länge
	fLength: LREAL;
	///Breite
	fWidth: LREAL;
	///Dicke
	fHeigth: LREAL;
	/// @1: maschinenspezifische Daten @11:2
	arrMaschine: ARRAY[1..2] OF ST_HMIPDatMaschine;
	///@1: Handfunktionen @6:1  @11:1
	manualFuntction: ST_HMI_Manual;
	///@1: Handfunktionen2 @6:1  @11:1
	manualFuntction2: ST_HMI_Manual; 
 
END_STRUCT
END_TYPE

// ---- Data types/MaschinenDaten PlcStructure/ST_PDatLineProgLine.TcDUT
TYPE ST_PDatLineProgLine :
STRUCT
	/// @1:Verechung der Teilelaenge/Breite in den Streckenwerkzeugen @11:2
	nSpezModus: INT;
	/// @1: Schaltmodus @11:2
	nSchaltmodus: INT;
	/// @1: Schaltkante ein @11:2
	nSchaltkanteEin: INT;
	/// @1: Schaltkante aus @11:2
	nSchaltkanteAus: INT;
	/// @1: Korrektur Schaltwert ein 				@2:mm @11:2
	fKorrSchaltwertEin: LREAL; 
	/// @1: Korrektur Schaltwert aus 				@2:mm @11:2
	fKorrSchaltwertAus: LREAL;
	///	@1: Korrektur Impluslänge 					@2:mm @11:2
	fKorrImpulslaenge: LREAL;
	/// @1: Korrektur Reaktionszeit Einsetzen 	@2:s @11:2
	fKorrReaktionszeitEinsetzen: LREAL;
	/// @1: Korrektur Reaktionszeit Aussetzen 	@2:s @11:2
	fKorrReaktionszeitAussetzen: LREAL;
END_STRUCT
END_TYPE

// ---- Data types/MaschinenDaten PlcStructure/ST_PDatLineProgValue.TcDUT
TYPE ST_PDatLineProgValue :
STRUCT
	///@1: StringWerte @11:2
	sValue: ARRAY[1..5] OF STRING(25);
	///@1: IntWerte @11:2
	nValue: ARRAY[1..5] OF INT;
	///@1: LrealWerte @11:2
	fValue: ARRAY[1..5] OF LREAL;
END_STRUCT
END_TYPE

// ---- Data types/Recipe/RecipeHeader_Struct.TcDUT
TYPE RecipeHeader_Struct :
STRUCT
	/// PLC -> HMI 
	RezeptAnf: STRING(40);
	/// HMI -> PLC 
	RezeptAkt: STRING(40);
	sReserve: ARRAY[3..10] OF STRING(40);
	Values: ARRAY[1..30] OF LREAL;
	List: ARRAY[1..50] OF RecipeList_Struct;
END_STRUCT
END_TYPE

// ---- Data types/Recipe/RecipeList_Struct.TcDUT
TYPE RecipeList_Struct :
STRUCT
	ToolId: LREAL;
	PosX: LREAL;
	PosY: LREAL;
	PosZ: LREAL;
	Tool1: LREAL;
	Tool2: LREAL;
	Tool3: LREAL;
	GlueTime: LREAL;
	Velo: LREAL;
	Reserve: ARRAY[10..20] OF LREAL;
END_STRUCT
END_TYPE

// ---- Data types/SERCOS/E_SoE_AttribLen.TcDUT
TYPE E_SoE_AttribLen :
(
	eSoE_LEN_2BYTE := 1,
	eSoE_LEN_4BYTE := 2,
	eSoE_LEN_8BYTE := 3,
	eSoE_LEN_V1BYTE := 4,
	eSoE_LEN_V2BYTE := 5,
	eSoE_LEN_V4BYTE := 6,
	eSoE_LEN_V8BYTE := 7
);
END_TYPE

// ---- Data types/SERCOS/E_SoE_CmdControl.TcDUT
TYPE E_SoE_CmdControl :
(
	eSoE_CmdControl_Cancel := 0,
	eSoE_CmdControl_Set := 1,
	eSoE_CmdControl_SetAndEnable := 3
);
END_TYPE

// ---- Data types/SERCOS/E_SoE_CmdState.TcDUT
TYPE E_SoE_CmdState :
(
	eSoE_CmdState_NotSet := 0,
	eSoE_CmdState_Set := 1,
	eSoE_CmdState_Executed := 2,
	eSoE_CmdState_SetAndInterrupted := 5,
	eSoE_CmdState_SetEnabledNotExecuted := 7,
	eSoE_CmdState_Error := 15
);
END_TYPE

// ---- Data types/SERCOS/E_SoE_Type.TcDUT
TYPE E_SoE_Type :
(
	eSoE_Type_BIN := 0,
	eSoE_Type_UNSIGNED := 1,
	eSoE_Type_SIGNED := 2,
	eSoE_Type_HEX := 3,
	eSoE_Type_TEXT := 4,
	eSoE_Type_IDN := 5,
	eSoE_Type_FLOAT := 6
);
END_TYPE

// ---- Data types/ST_Diagnose.TcDUT
TYPE ST_Diagnose :
STRUCT
	Hydraulik: FB_Diag;
	Pneumatik: FB_Diag;
	Kuehlung: FB_Diag;
	MSGList1: ARRAY[FIRST_MESSAGE..LAST_MESSAGE] OF BOOL;
	MSGListQuit1: ARRAY[FIRST_MESSAGE..LAST_MESSAGE] OF BOOL;
	MSGList2: ARRAY[FIRST_MESSAGE..LAST_MESSAGE] OF BOOL;
	MSGListQuit2: ARRAY[FIRST_MESSAGE..LAST_MESSAGE] OF BOOL;
END_STRUCT
END_TYPE

// ---- Data types/ST_EtherCATAxisInfo.TcDUT
TYPE ST_EtherCATAxisInfo :
STRUCT
	NetId: STRING(MAX_STRING_LENGTH);
	id: DINT;
	nCha: UINT;
	nPort: UINT;
	stDriveRef: ST_SoE_DriveRef;
END_STRUCT
END_TYPE

// ---- Data types/ST_EventData1.TcDUT
TYPE ST_EventData1 :
STRUCT
	axis: UDINT;
	pos: LREAL;
END_STRUCT
END_TYPE

// ---- Data types/ST_EventDataAX5000_1.TcDUT
TYPE ST_EventDataAX5000_1 :
STRUCT
	nDiagNumber: UDINT;
	nAxisId: UDINT;
	sChannel: STRING(120);
END_STRUCT
END_TYPE

// ---- Data types/ST_MachineMode.TcDUT
TYPE ST_MachineMode :
STRUCT
	/// Operation Mode 
	Standby: BOOL;
	Manual: BOOL;
	MDI: BOOL;
	Automatic: BOOL;
	///REFERENCE		: BOOL;  TC3HR
	Homing: BOOL;
	/// Operation State
	Select : BOOL; 
	Ready  : BOOL;
	Start: BOOL;
	Stop: BOOL;
	Reset: BOOL;
	Error: BOOL;
	/// Special functions 
	ChannelSignals: ST_ChannelSignals;
	BlockSearch: ST_BlockSearch;
	SyntaxCheck: ST_SyntaxCheck;
	ManualMode: ST_ManualMode;
	/// Strings 
	ProgramName: STRING(1024);
	MDIString: STRING(1024);
END_STRUCT
END_TYPE

// ---- Data types/ST_MViewStatus.TcDUT
TYPE ST_MViewStatus :
STRUCT
	Color: ARRAY[1..MV_NUMBER_OF_ROWS] OF INT;
	Description: ARRAY[1..MV_NUMBER_OF_ROWS] OF STRING(80);
END_STRUCT
END_TYPE

// ---- Data types/ST_WKZDaten.TcDUT
TYPE ST_WKZDaten :
STRUCT
	nAblageX: LREAL;
	nAblageY: LREAL;
	nWkzLaenge: LREAL;
	nWkzRadius: LREAL;
	nStandzeit: LREAL;
	nStandWeg: LREAL;
	nReserve: ARRAY[7..40] OF LREAL;
END_STRUCT
END_TYPE

// ---- Data types/ST_WPCounter.TcDUT
TYPE ST_WPCounter :
STRUCT
	CompleteCounterAll: DINT;
	CompleteCounterIO: DINT;
	CompleteCounterNIO: DINT;
	DailyCounterAll: DINT;
	DailyCounterIO: DINT;
	DailyCounterNIO: DINT;
	ShiftCounterAll: DINT;
	ShiftCounterIO: DINT;
	ShiftCounterNIO: DINT;
END_STRUCT
END_TYPE

// ---- Global Variables/Examples/Globale_EtherCATDiag.TcGVL
VAR_GLOBAL CONSTANT
	iSLAVEADDR_ARR_SIZE: INT := 255;
END_VAR

// ---- Global Variables/Examples/Global_BDE.TcGVL
VAR_GLOBAL
	///--------------------------
	///	BDE, PLC -> HMI          
	///--------------------------
	BDESteuerungEin: BOOL;
	BDEAutomatik: BOOL;
	BDEVarBoolTimer: ARRAY[0..10] OF BOOL;
	BDEVarBoolCounter: ARRAY[0..10] OF BOOL;
	BDEVarBoolMessage: ARRAY[0..50] OF BOOL;
END_VAR

// ---- Global Variables/Examples/Global_MachineView.TcGVL
VAR_GLOBAL CONSTANT
	///--------------------------
	///	Machine View Status      
	///--------------------------
	MV_NUMBER_OF_ROWS: INT := 6;
	/// dynamically no maximum 
	MV_NUMBER_OF_BLOCKS: INT := 4;
END_VAR

VAR_GLOBAL
	MViewStatus: ARRAY[1..MV_NUMBER_OF_BLOCKS] OF ST_MViewStatus;
END_VAR

// ---- Global Variables/Examples/Global_ManualPlcFunctions.TcGVL
VAR_GLOBAL
	
	PortalInfo			: STRING;
	PortalOn			: ARRAY[1..20] OF BOOL;
	PortalOff			: ARRAY[1..20] OF BOOL;
	PortalStatus		: ARRAY[1..20] OF BYTE;
	
	HandAnwInfo			: STRING;
	HandAnwOn			: ARRAY[1..20] OF BOOL;
	HandAnwOff			: ARRAY[1..20] OF BOOL;
	HandAnwStatus		: ARRAY[1..20] OF BYTE;
END_VAR

// ---- Global Variables/Examples/Global_MaschinenDaten.TcGVL
VAR_GLOBAL CONSTANT
	MAX_TOOLS: INT := 20;
	MAX_WKZLIMITS: INT := 25;
	MAX_TIMER: INT := 50;
	/// BDE - Meldungen 
	BDE_MSG_1: INT := 1;
	BDE_MSG_2: INT := 2;
	BDE_MSG_3: INT := 3;
	/// BDE - Timer 
	BDE_TIMER_SUMME: INT := 1;
	BDE_TIMER_STEUERUNGEIN: INT := 2;
	BDE_TIMER_AUTOMATIK: INT := 3;
	BDE_TIMER_STOERUNG: INT := 4;
	/// BDE - Counter 
	BDE_COUNTER_AUTO: INT := 1;
	BDE_COUNTER_STUECKZAHL: INT := 2;
	/// Allgemeine Maschinendaten Offsets 
	MASCH_GRUNDPOS_ACHSE_X: INT := 1;
	MASCH_GRUNDPOS_ACHSE_Y: INT := 2;
	MASCH_GRUNDPOS_ACHSE_Z: INT := 3;
	MASCH_GRUNDPOS_ACHSE_L: INT := 4;
	MASCH_GRUNDPOS_ACHSE_o: INT := 4;
END_VAR

VAR_GLOBAL

	///@1:Maschinendaten
	MachData: ST_MachData;  

	bStartWriteFromHMI: BOOL;
	bWriteReadyFromHMI: BOOL;
	bReadFromPlc: BOOL;
	sFileName: STRING(255);
	///--------------------------
	///	Maschinendatentabellen  
	///--------------------------
	PLCMParList1: ARRAY[1..101] OF LREAL;
	PLCMParList2: ARRAY[1..101] OF LREAL;
	PLCMParList3: ARRAY[1..50] OF LREAL;
	/// Tooldata 
	WkzWechslerPos1: ARRAY[1..41] OF LREAL;
	/// position in tool changer in the order x1,y1,z1a,z1b,x2,y2,z2a,z2b.... 
	WkzWechslerPos2: ARRAY[1..41] OF LREAL;
	/// position in tool changer in the order x1,y1,z1a,z1b,x2,y2,z2a,z2b.... 
	WkzWechslerPos3: ARRAY[1..41] OF LREAL;
	aktTool: ST_CNC_TOOL_DATA_EXT;
	oldTool: ST_CNC_TOOL_DATA_EXT;
	/// ID of requested Tool Data 
	nToolRequestID: DINT;
	/// Sister ID of requested Tool Data, ignored if 0
	nToolRequestIDSister: DINT;
	/// with rising edge -> start transfer HMI -> PLC (aktTool), falling edge -> HMI reports done 
	bToolData: BOOL;
	/// with rising edge -> data is transfered PLC -> HMI, falling edge -> HMI reports done 
	bOldToolData: BOOL;
	/// Timer 
	PLCTimer: ARRAY[1..MAX_TIMER] OF REAL;
	/// Geschwindigkeiten 
	GeschwLeer: ARRAY[1..10] OF REAL;
	GeschwLast: ARRAY[1..10] OF REAL;
	/// Allgemeine Maschinendaten 
	MaschParam: ARRAY[1..50] OF REAL;
	TestBol: ARRAY[1..50] OF BOOL;
	/// HMi -> PLC set to true, after writing all Maschpara 
	bWriteToPlc: BOOL;
	/// aktual Tool ID of tool in CNC 
	nToolInCnc: DINT;
	nToolInCncSister: DINT;
	VE_Tool: UINT;
	dwtest: DWORD;
END_VAR

// ---- Global Variables/Examples/Global_VE.TcGVL
VAR_GLOBAL
	PLC_OffsetX: LREAL := 123.23;
	PLC_OffsetY: LREAL := 223.23;
	PLC_OffsetZ: LREAL := 323.23;
	/// HMI -> PLC 
	HMI_PLC_OffsetX: LREAL;
	HMI_PLC_OffsetY: LREAL;
	HMI_PLC_OffsetZ: LREAL;
END_VAR

// ---- Global Variables/Global_CNC.TcGVL
VAR_GLOBAL
	CNCSystem						: ST_CncSystem;
END_VAR

(****************************************************************************************)
(*	  	Global constants used by the fast M function handling process (MOS_TS)			*)
(****************************************************************************************)
VAR_GLOBAL CONSTANT
	MAX_FAST_M_FUNC_ITEM_IDX	: UINT	:= 7;			(* Max. index of fast M functions processed by HLI3_FastMFunctionProvider per PLC cycle *) 
	MAX_FAST_M_FUNC_QUEUE_IDX	: UINT	:= 63;			(* Max. index of fast M function switch events buffered by HLI3_FastMFunctionHandler *) 
	MAX_FAST_M_FUNC_OUTPUT_IDX	: UINT	:= 124;			(* Max. index of fast M function oversampling output byte array *)			
	MAX_SYS_LOG_AXIS_INDEX		: UINT  := 255;			(* Max. Index of Log. Axis Id *) 				
	
	MAX_USED_CHANNEL_IDX		: INT := 0;				(* Max index of channel that is used starting at 0, example: 1 -> totally 2 channels, maximum of 11 (12 channels) is allowed here *)
	
	stVersion_CNCPlcBaseProject : ST_LibVersion := STRUCT(iMajor := 3, iMinor := 1, iBuild := 3035, iRevision := 30, sVersion := '3.1.3035.30');
END_VAR

// ---- Global Variables/Global_CNCVariablesViewer.TcGVL
{attribute 'pack_mode' := '1'}
VAR_GLOBAL
	stCNCVariablesViewer_Data : ARRAY[0..MAX_CNC_VAR_LIST_IDX] OF ST_CNCVariablesViewer_Data;
	eVariablesType : E_CNCVariablesType;

END_VAR

VAR_GLOBAL CONSTANT
	MAX_CNC_VAR_LIST_IDX : UINT := 200;
END_VAR

// ---- Global Variables/Global_HMI.TcGVL
VAR_GLOBAL
	/// HMI -> PLC 
	PLCChannelSignals: ST_ChannelSignals;
	/// HMI -> PLC 
	PLCSelectedChannel: INT := 1;
	/// HMI -> PLC 
	PLCFeedOverride: UINT := 100;
	/// HMI -> PLC 
	PLCSpindleOverride: UINT := 100;
	/// HMI -> PLC 
	PLCAxisEnable: BOOL;
	/// HMI -> PLC 
	PLCReset: BOOL;
	PLCMachineMode: ARRAY[0..MAX_USED_CHANNEL_IDX+1] OF ST_MachineMode;
	/// PLC -> HMI : angewähltes File 
	PLCToHmiFile: STRING(255);
	/// Variablen für das Module "InformPlc" 
	bToggle: BOOL;
	sActualForm: STRING(255);
	nUserLevel: INT;
	sUserName: STRING(255);
	/// steigende Flanke: Applikation beenden 
	bExitApp: BOOL;	
	
	userActivity : BOOL;
	
	TimeTest: TIME := T#1250MS;
	
	(*stat: EventStatistik; *)
END_VAR

// ---- Global Variables/Global_ManualMode.TcGVL
VAR_GLOBAL
/// Selection of manual mode controller 
	geManualModeController: E_CNC_MM_Controller;
	/// Manual mode control structures 
	stManualModeParameter: ARRAY[0..11] OF ST_ManualModeParameter;
	stManualModeControlElements: ARRAY[0..11] OF ST_ManualModeControlElements;
	stManualModeState: ARRAY[0..11] OF ST_ManualModeState;
	stManualModeControlElementState : ST_ManualModeControlElementState;
END_VAR

// ---- Global Variables/Global_Messages.TcGVL
VAR_GLOBAL
	///--------------------------
	///	Messages                
	///--------------------------
	MSG_WARNING_List: ARRAY[FIRST_MESSAGE..LAST_MESSAGE] OF BOOL;
	MSG_WARNING_ListQuit: ARRAY[FIRST_MESSAGE..LAST_MESSAGE] OF BOOL;	
	MSG_ALARM_List: ARRAY[FIRST_MESSAGE..LAST_MESSAGE] OF BOOL;
	MSG_ALARM_ListQuit: ARRAY[FIRST_MESSAGE..LAST_MESSAGE] OF BOOL;	
END_VAR

VAR_GLOBAL CONSTANT
	FIRST_MESSAGE: UDINT := 1;
	LAST_MESSAGE: UDINT := 50;
	FIRST_SYSTEM_MESSAGE: UDINT := 1;
	LAST_SYSTEM_MESSAGE: UDINT := 10;
	nSourceTextPtpNci: UINT := 700;
	nSourceDescPtpNci: UINT := 701;
	nSourceChannel: UINT := 702;
	nSourceAxis: UINT := 800;
	nSourcePlc: UINT := 1100;
	nEventChannel: UINT := 200;
	nEventAxis: UINT := 201;
	nEventPlc: UINT := 202;
END_VAR

// ---- Global Variables/Variable_Configuration.TcGVL
VAR_GLOBAL
END_VAR

// ---- Version/Global_Version.TcGVL
{attribute 'TcGenerated'}
// This function has been automatically generated from the project information.
VAR_GLOBAL CONSTANT
	{attribute 'const_non_replaced'}
	{attribute 'linkalways'}
	stLibVersion_CNC_PLC_Project : ST_LibVersion := (iMajor := 3, iMinor := 1, iBuild := 3035, iRevision := 30, sVersion := '3.1.3035.30');
END_VAR

// ---- FAST.TcPOU
PROGRAM FAST
VAR
	nChan : INT;
	MOS_TS: INT;
END_VAR

(****************************************************************************************)
(*	  							Wait for HLI initialization								*)
(****************************************************************************************)
IF NOT CNCSystem.bHLIInit THEN
	RETURN;
END_IF

(* Programm call for MOS_TS M functions *)
// PRG_FastMFunctions();

(* CNC Watchdog mechanism *)
FOR nChan := 0 TO MAX_USED_CHANNEL_IDX DO
	IF (HLI3_CheckChannelValid(nChan)) THEN	
		HLI3_SetPLCAlive(nChanIdx :=  nChan);
		//HLI3_CheckCNCAlive(nChanIdx := nChan);
	END_IF
END_FOR

END_PROGRAM

// ---- CNC Beckhoff/9 Mis/HLI3_CheckChannelValid.TcPOU
FUNCTION HLI3_CheckChannelValid : BOOL
VAR_INPUT
	nChannel: INT;
END_VAR

(* ========================================================= *)
(*    FUN: HLI3_CheckChannelValid                            *)
(* --------------------------------------------------------- *)
(*   Desc: Check if channel ID is valid for HLI access       *)
(*   Author: MiB                                             *)
(*   Date: 19.11.2012                                        *)
(*   Last: 21.06.2013										 *)
(*   Rev.: 1.1                                               *)
(* --------------------------------------------------------- *)
(*   Desc: Corrected IF statement (line 14)		 	      	 *)
(*   Author: RCH                                             *)
(*   Date: 16.09.2013                                        *)
(*   Rev.: 1.2                                               *)
(* ========================================================= *)

IF (nChannel < 0) THEN
	HLI3_CheckChannelValid:= FALSE;
	RETURN; (* A b b r u c h *)
ELSIF (nChannel >=  UDINT_TO_INT(gNrCh) ) OR		(* check for channel no *)
       (gpCh[nChannel] = 0) 				  (* check for zero pointer *)
THEN
	HLI3_CheckChannelValid:= FALSE;
	RETURN; (* A b b r u c h *)
ELSE
	HLI3_CheckChannelValid := TRUE;
	RETURN;
END_IF

END_FUNCTION

// ---- CNC Beckhoff/9 Mis/HLI3_SetPLCAlive.TcPOU
FUNCTION HLI3_SetPLCAlive : BOOL
VAR_INPUT
	nChanIdx: INT;
END_VAR

(*
Display PLC is just alive (Trigger Watchdog to MC)
If PLC is stopped here, alive sign is missing.
-> CNC raises error message
-> CNC stoppes movement with internal FEEDHOLD
-> system has to be restarted (after removal of error)
*)

HLI3_SetPLCAlive := FALSE;
IF NOT HLI3_CheckChannelValid(nChannel := nChanIdx) THEN
	RETURN;
END_IF

gpCh[nChanIdx]^.head.mc_watchdog.enable_w := TRUE;
gpCh[nChanIdx]^.head.mc_watchdog.alive_rw := TRUE;

HLI3_SetPLCAlive := TRUE;

END_FUNCTION

// ---- MAIN.TcPOU
PROGRAM MAIN
VAR	
	ZyklenString:STRING;
	Trennscheibe AT %Q*:INT;
	DigitalIn AT %I*:INT;
	temp:bool;
END_VAR
VAR PERSISTENT
	ZyklenInt:LINT;
END_VAR

(****************************************************************************************)
(* POU:		MAIN                     													*)
(* Type:	PRG																			*)
(* Author: 	HR , TV                                              						*)
(* Date: 	24.01.11																	*)
(* Last:	21.01.14																*)
(* Rev.: 	1.02                                               							*)
(* ------------------------------------------------------------------------------------ *)
(* Desc:	Main program frame for CNC sample applications								*)
(****************************************************************************************)

(****************************************************************************************)
(*								Infrastructure programs									*)
(****************************************************************************************)
PRG_ShowMessages();
(****************************************************************************************)
(*										CNC programs									*)
(****************************************************************************************)
HLI3_Init(); 
(* Call CNC related code only if the HLI has been initialized succesfully! *)
IF CNCSystem.bHLIInit THEN
	PRG_AxesHandler();    	
	PRG_ManualMode();  
	PRG_ChannelHandler();
	PRG_CNCVariablesViewer();
END_IF

(* Reset the reset flag from HMI *)
PLCReset := FALSE;

IF Global_CNC.CNCSystem.Channel[0].M[99].bState_rw THEN
	Global_CNC.CNCSystem.Channel[0].M[99].bState_rw:=FALSE;
	ZyklenInt:=ZyklenInt+1;
	ZyklenString:=LINT_TO_STRING(ZyklenInt);
END_IF

IF Global_CNC.CNCSystem.Channel[0].M[100].bState_rw THEN
	Global_CNC.CNCSystem.Channel[0].M[100].bState_rw:=FALSE;
	ZyklenInt:=0;
	ZyklenString:=LINT_TO_STRING(ZyklenInt);
END_IF

IF Global_CNC.CNCSystem.Channel[0].M[101].bState_rw THEN
	Global_CNC.CNCSystem.Channel[0].M[101].bState_rw:=FALSE;
	Trennscheibe:=128;
END_IF
IF Global_CNC.CNCSystem.Channel[0].M[102].bState_rw THEN
	Global_CNC.CNCSystem.Channel[0].M[102].bState_rw:=FALSE;
	Trennscheibe:=0;
END_IF
temp:=GETBIT32(DigitalIn,6);
IF NOT temp AND Global_CNC.CNCSystem.Channel[0].ActState=4 THEN
	PLCMachineMode[1].Error:=TRUE;
	PLCMachineMode[1].Stop:=true;
END_IF
PLCMachineMode[1].Stop:=false;

END_PROGRAM

// ---- CNC Beckhoff/PRG_ShowMessages.TcPOU
PROGRAM PRG_ShowMessages
VAR
	bStart: BOOL;
	fbWarningMessages : FB_SimpleEventLog;
	fbAlarmMessages : FB_SimpleEventLog;
END_VAR

(*
	TCEVENTCLASS_NONE			:=0,	 No class
	TCEVENTCLASS_MAINTENANCE	:=1,	 Maintenance hint
	TCEVENTCLASS_MESSAGE		:=2,	 Message
	TCEVENTCLASS_HINT			:=3,	 Hint
	TCEVENTCLASS_STATEINFO		:=4,	 State information
	TCEVENTCLASS_INSTRUCTION	:=5,	 Instruction
	TCEVENTCLASS_WARNING		:=6,	 Warning
	TCEVENTCLASS_ALARM			:=7,	 Alarm
	TCEVENTCLASS_PARAMERROR		:=8	 Parameter error
*)


(* Shows how to generate messages *)
IF NOT bStart THEN
	bStart 				:= TRUE;

	fbWarningMessages
		(Init			:= TRUE,
		 SourceId		:= 51,
		 Class			:= TCEVENTCLASS_WARNING,
		 QuitRequireD	:= FALSE,
		 adrAlarmArray	:= ADR(MSG_WARNING_List),
		 adrQuitArray	:= ADR(MSG_WARNING_ListQuit)
		);

	fbAlarmMessages
		(Init			:= TRUE,
		 SourceId		:= 50,
		 Class			:= TCEVENTCLASS_ALARM,
		 QuitRequired	:= FALSE,
		 adrAlarmArray 	:= ADR(MSG_ALARM_List),
		 adrQuitArray	:= ADR(MSG_ALARM_ListQuit)
		);
ELSE
	fbWarningMessages
		(Init			:= FALSE);

	fbAlarmMessages
		(Init			:= FALSE);	
END_IF

END_PROGRAM

// ---- CNC Beckhoff/Messages/FB_SimpleEventLog.TcPOU
///****************************************************************************************
///Name:				FB_SimpleEventLog
///Date:				13.10.2004
///Author:			Dirk Nordberg (BECKHOFF INDUSTRIE ELEKTRONIK)
///
///Description: Function block to control the EventLogger
///	Messages can be activated or deactivated through an array of bool.
///	The subscription of the array is equivalent to EventID from EventLogger.
///	Funtion block will be initialized with Init flag, then the busy flag is set true. 
///
///	Revision:	1.4
///	History:		13.10.2004	Ng	start coding
///					17.04.2005	MK	runtime optimized
///					07.07.2005	MK	short puls BF
///				    29.11.2010 	MiB  quittierungspflichtige Merker funktionieren nun wieder
///                 21.06.2013  TV   change : data type for pointer address from uint to pointer of int 
///****************************************************************************************
FUNCTION_BLOCK FB_SimpleEventLog
VAR_INPUT
	/// Rising flag starts the initialization 
	Init: BOOL;
	/// Number of the source Id 
	SourceId: UINT;
	/// Alarm error class 
	Class: UINT;
	/// Activate or deaktivate confirmation 
	QuitRequired: BOOL;
	/// Adress of the array for the messages 
	adrAlarmArray: POINTER TO BOOL;
	/// ...with constant boundaries ARRAY_LBOUND to ARRAY_UBOUND for array size 
	adrQuitArray: POINTER TO BOOL;
END_VAR
VAR_OUTPUT
	Busy: BOOL;
	Err: BOOL;
	ErrId: UDINT;
END_VAR
VAR CONSTANT
	ARRAY_LBOUND: UDINT := FIRST_MESSAGE;
	ARRAY_UBOUND: UDINT := LAST_MESSAGE;
	TCEVENTDATAFORMATSTRING: STRING := ' ';
	STATE_INIT: INT := 0;
	STATE_IDLE: INT := 1;
	STATE_RESET_EVENT: INT := 2;
	STATE_QUIT_EVENT: INT := 3;
	STATE_RESET_END: INT := 4;
	STATE_WAIT: INT := 5;
END_VAR
VAR
	state: INT;
	///{flag nowatch on }
	bReady: BOOL := TRUE;
	nMsgHasChanged: DINT;
	bEvtState: ARRAY[ARRAY_LBOUND..ARRAY_UBOUND] OF BOOL;
	event: ARRAY[ARRAY_LBOUND..ARRAY_UBOUND] OF ADSLOGEVENT;
	idx: UDINT;
	CfgEvent: TcEvent;
	bWait: BOOL;
	ptAlarm: POINTER TO BOOL;
	ptQuit: POINTER TO BOOL;
	RT_Init: R_TRIG;
END_VAR

nMsgHasChanged := MEMCMP(ADR(bEvtState), adrAlarmArray, SIZEOF(bEvtState));

RT_Init(CLK:=Init);

CASE State OF
	STATE_INIT:		(* Set the parameter for TcEvent *)
		Err := FALSE;
		ErrId :=0;
		Busy := FALSE;
		CfgEvent.Prio := 0;
		CfgEvent.DataFormatStrAddress := ADR(TCEVENTDATAFORMATSTRING);
		// CfgEvent.Flags := TCEVENTFLAG_LOG OR TCEVENTFLAG_SRCID OR TCEVENTFLAG_PRIOCLASS OR TCEVENTFLAG_FMTSELF OR 16#1000;
		// MiB 2015.10.07 Flags changed -> now the class is defined here and not in Event config file.
		CfgEvent.Flags := TCEVENTFLAG_LOG OR TCEVENTFLAG_SRCID;
		CfgEvent.StreamType := TCEVENTSTREAM_SIMPLE;
		CfgEvent.ProgId := 'TcEventFormatter.TcXmlFormatter';
		CfgEvent.SourceId := SourceId;
		CfgEvent.Class := Class ;
		CfgEvent.bQuitRequired := QuitRequired;
		FOR idx := ARRAY_LBOUND TO ARRAY_UBOUND BY 1 DO
			CfgEvent.Id := idx;
			event[idx](NETID:='', PORT:=110, Event:=FALSE , EventQuit:=FALSE,
				 EventConfigData:=CfgEvent, FbCleanup:=FALSE, TMOUT:=t#1s);
		END_FOR;
		State := STATE_IDLE;

	STATE_IDLE:
		(* nothing to do *)
		IF nMsgHasChanged = 0
			AND  NOT QuitRequired
			AND bReady = TRUE
			AND NOT RT_Init.Q THEN
			RETURN;
		END_IF

		IF adrAlarmArray <> 0 THEN
			ptAlarm := adrAlarmArray;
			IF CfgEvent.bQuitRequired AND adrQuitArray <> 0 THEN
				ptQuit := adrQuitArray;
				FOR idx := ARRAY_LBOUND TO ARRAY_UBOUND BY 1 DO
					event[idx](Event:=ptAlarm^, EventQuit:=ptQuit^);
					ptAlarm := ptAlarm + 1;
					ptQuit := ptQuit + 1;
				END_FOR;
				bReady := TRUE;
			ELSE
				bReady := TRUE;
				FOR idx := ARRAY_LBOUND TO ARRAY_UBOUND BY 1 DO
					event[idx](Event:=ptAlarm^);
					IF (NOT (ptAlarm^ = TRUE
							AND event[idx].Event = TRUE		(* event is set/on *)
							AND event[idx].Quit = FALSE
							AND event[idx].EventState = TCEVENTSTATE_SIGNALED)
						AND NOT (ptAlarm^ = FALSE
							AND event[idx].Event = FALSE		(* event is reset/off *)
							AND event[idx].Quit = TRUE
							AND event[idx].EventState = TCEVENTSTATE_INVALID)) THEN
						bReady := FALSE;
					END_IF
					ptAlarm := ptAlarm + 1;
				END_FOR;

				(* copy the status *)
				IF bReady THEN
					MEMCPY(ADR(bEvtState), adrAlarmArray, SIZEOF(bEvtState));
				END_IF

			END_IF
		END_IF

		IF RT_Init.Q THEN
			Busy := TRUE;
			State := STATE_RESET_EVENT;
		END_IF

	STATE_RESET_EVENT:(*---------------------------------- clear messages ----------------------------------------*)
		FOR idx := ARRAY_LBOUND TO ARRAY_UBOUND BY 1 DO
			IF event[idx].EventState = TCEVENTSTATE_SIGNALED THEN
				event[idx](Event:=FALSE, EventQuit:= FALSE, FbCleanup:= FALSE, TMOUT:= t#1s);
				IF event[idx].Err THEN
					Err := TRUE;
					ErrId := event[idx].ErrId;
					IF event[idx].ErrId = 1282 THEN	(* Message Router: mailbox full *)
						event[idx](Event:=FALSE, EventQuit:= FALSE, FbCleanup:= FALSE);
						RETURN;
					END_IF
				END_IF
			END_IF;
		END_FOR;
		State := STATE_QUIT_EVENT;

	STATE_QUIT_EVENT:(*---------------------------------- quit messages ----------------------------------------*)
		FOR idx := ARRAY_LBOUND TO ARRAY_UBOUND BY 1 DO
			IF event[idx].EventState = TCEVENTSTATE_SIGNALED THEN
				event[idx](Event:=FALSE, EventQuit:= TRUE, FbCleanup:= FALSE, TMOUT:= t#1s);
				IF event[idx].Err THEN
					Err := TRUE;
					ErrId := event[idx].ErrId;
					IF event[idx].ErrId = 1282 THEN	(* Message Router: mailbox full *)
						event[idx](Event:=FALSE, EventQuit:= FALSE, FbCleanup:= FALSE);
						RETURN;
					END_IF
				END_IF
			END_IF;
		END_FOR;
		State := STATE_RESET_END;

	STATE_RESET_END:
		bWait := FALSE;
		FOR idx := ARRAY_LBOUND TO ARRAY_UBOUND BY 1 DO
			event[idx](Event:=FALSE, EventQuit:= FALSE, FbCleanup:= FALSE);
			IF event[idx].EventState = TCEVENTSTATE_SIGNALED THEN
				bWait := TRUE;
			END_IF
		END_FOR;
		IF NOT bWait THEN
			State := STATE_INIT;
		END_IF

END_CASE

END_FUNCTION_BLOCK

// ---- CNC Beckhoff/1 Init/HLI3_Init.TcPOU
PROGRAM HLI3_Init
VAR
	Hli: MCV_HliInterface;
	bFirstCycle: BOOL := TRUE;
	ipSrv: ITComObjectServer;
	oidCnc: UDINT := 16#5500001;
	bUnregister: BOOL;
	MessageOutput: R_TRIG;
	nHliAxisIdx	: INT;
END_VAR

(* ========================================================= *)
(*    PRG: HLI_Init                                          *)
(* --------------------------------------------------------- *)
(*   Desc:                                                   *)
(* Author: MK                                                *)
(*   Date: 21.12.2011                                        *)
(*   Rev.: 1.0                                               *)
(*   Date: 06.08.2013                                        *)
(*   Rev.: 1.1 TV   Error Message if HLI not initialized	 *)
(* ========================================================= *)


(* Init Tool Configuration structures *)
HLI3_InitToolConfig();

IF bFirstCycle THEN
	Hli();					(* initialize HLI *)
	bFirstCycle := FALSE;
END_IF


IF Hli.Initialized  = TRUE
THEN
	(* User initialization, used during start of PLC once *)
	IF CncSystem.bUserInitDone = FALSE THEN
		(* Initialisierungen auf dem HLI-Interface *)
		CncSystem.bUserInitDone := HLI3_UserInitialisation();
		ADSLOG(strMsg:='High Level Interfaces initialized: %s', nDINT:=0, strArg:='');
	END_IF

	IF (NOT CNCSystem.bHLIInit) THEN
		FOR nHliAxisIdx := 0 TO HLI_SYS_AX_MAXIDX DO
        	IF HLI3_CheckAxisValid(nHliAxisIdx) THEN
            	CNCSystem.LogAxisNo[gpAx[nHliAxisIdx]^.ipo_state.log_achs_nr_r].nHliAxisIdx := nHliAxisIdx;
                CNCSystem.LogAxisNo[gpAx[nHliAxisIdx]^.ipo_state.log_achs_nr_r].stLogName   := gpAx[nHliAxisIdx]^.lr_state.log_name_r.zeichen;                          
           	END_IF
		END_FOR
	END_IF
	
	(* initialization finished *)
	CNCSystem.bHLIInit := TRUE;
ELSE
	MessageOutput(CLK:=Hli.Error);
	IF Hli.Error = TRUE	THEN
		(* High Level Interface (HLI) not initialized *)
		IF MessageOutput.Q THEN
			ADSLOGDINT(	msgCtrlMask := ADSLOG_MSGTYPE_ERROR OR
												ADSLOG_MSGTYPE_MSGBOX OR
												ADSLOG_MSGTYPE_LOG,
							msgFmtStr := 'High Level Interface (HLI) not initialized! Errorcode: %d',
							dintArg := Hli.ErrorID);
		END_IF
		CNCSystem.nInitErrorId := Hli.ErrorID;
		CNCSystem.bInitError := TRUE;
	END_IF;	
END_IF

END_PROGRAM

// ---- CNC Beckhoff/1 Init/HLI3_InitToolConfig.TcPOU
PROGRAM HLI3_InitToolConfig
VAR
	BasicToolId: DINT;
	pToolId: POINTER TO CNC_TOOL_ID;
	pToolReq: POINTER TO CNC_TOOL_REQUEST_IN;
	pToolLife: POINTER TO CNC_TOOL_DATA_IN;
	Rind: ADSRDWRTIND;
	RRes: ADSRDWRTRES;
	bRes: BOOL;
	i: INT;
	nr: DINT;
	SisterToolID: DINT;
	d1: UINT;
	t1: UINT;
	fbRTrigD: R_TRIG;
	fbRTrigOldData: R_TRIG;
	T0: CNC_TOOL_DATA;
	pos: INT;
	cnc_channel_nr: UDINT;
END_VAR

(* ---------------------*----------------------------------|------------------------------------------------------- *)
(* PURPOSE: External Tool Change                                                                                    *)
(*          used for tool change and tool live                                                                      *)
(*                                                                                                                  *)
(* SCOPE:                                                                                                           *)
(*                                                                                                                  *)
(*                                                                                                                  *)
(* REMARKS:                                                                                                         *)
(*                                                                                                                  *)
(*                                                                                                                  *)
(* AUTHOR:              VERSION     DATE                   CHECKED FROM      DATE     STATUS                        *)
(*    MK                1.0         07.05.2003                                                                      *)
(*    MiB               1.1         04.04.2006                                                                      *)
(*    MK                1.2         04.08.2006                                                                      *)
(*	  MiB					1.3			04.12.2006																						    	  *)
(*	  MiB					1.4			19.11.2012          TC3																					  *)
(*	  MiB					1.5			05.03.2015          TC3	  Zusatzparameter P[i]  werden aus der CNC zur PLC in OldTool übertragen		  *)
(*                                                                                                                  *)
(* ---------------------*----------------------------------|------------------------------------------------------- *)

(*
 ATTENTION: These Indications are only sent by the CNC if the CNC channel is configured accordingly:
In the SDA-MDS parammeter list the following parameters must be set:
- ext_wzv_vorhanden    1   -> (external tool managment present) Tool requests D<i> are sent TO external tool data manager
- einrechnen_mit_t     0/1 -> programming T<i> implies a programmed D<i>
- tool_life_to_wzv     1   -> send tool data life parameters TO external tool data manager IF tool is changed.
- t_info_to_wzv        1   -> send tool to external tool data manager IF tool is programmed.

CNC_TOOL_ID :
	basic					: DINT;
	sister				: DINT;
	variant				: DINT;
	sister_valid		: BOOL;
	variant_valid		: BOOL;
	res1					: BYTE;
	res2					: BYTE;
CNC_TOOL_REQUEST_IN :
	id						: CNC_TOOL_ID; 		(* tool id of requested tool *)
	act_t_nr				: DINT;					(* actual t number in nc kernel *)
	act_d_nr				: CNC_TOOL_ID; 		(* actual tool id (d-number) in the nc kernel *)
	param					: ARRAY [0..CNC_TOOL_PARAM_MAXIDX] OF LREAL;
CNC_TOOL_DESC :
	tool_id				: CNC_TOOL_ID;
	laenge				: DINT;
	radius				: DINT;
	ax_versatz			: ARRAY [0..CNC_TOOL_AXIS_OFFSET_MAXIDX] OF DINT;
	kopf_versatz		: ARRAY [0..CNC_TOOL_HEAD_OFFSET_MAXIDX] OF DINT;
	mass_einheit		: UINT;
	typ					: UINT;
	srk_lage			: UINT;
	kin_id				: UINT;
	log_ax_nr_spdl		: UINT;
	tool_fixed			: BOOL;
	valid				: BOOL;
	add_info			: ARRAY [0..HLI_ADD_INFO_MAXIDX] OF DWORD; (*additional tool information, can be used for fitting cycle *)
	res					: ARRAY [1..4] OF BYTE;
	param				: ARRAY [0..CNC_TOOL_PARAM_MAXIDX] OF LREAL;
	vb_min				: LREAL;
	vb_max				: LREAL;
	a_max				: LREAL;
*)


(* Init Tool Configuration *)
bRes := FALSE;
Rind();

IF PLCReset THEN
  	bToolData := FALSE;    (* Reset request to HMI *)
	bOldToolData := FALSE;
END_IF

IF Rind.VALID THEN
	(* initialize response *)
	RRes.NETID := '';
	RRes.PORT	:= Rind.PORT;
	RRes.INVOKEID := Rind.INVOKEID;

	(* sender channel nr is coded in the invoke id *) (* Kanalnummer zur Zeit nicht benutzt *)
	cnc_channel_nr := RInd.INVOKEID; 
	cnc_channel_nr := cnc_channel_nr AND 16#00FFFFFF; 
	
		
	(* Since there is only one ADSRDWRTIND possible per PLC task *)
	(* all indications have to be handled in one place *)
	(* To distinguish between several possible request types *)
	(* the indexgroup of the ADSRDWRTIND is used *)

	(*----- CNC tool data request with T<i>-----*)
	(* CNC teil den Werkzeugwechsel T<i> (während Programmdekodierung) mit *)
	IF Rind.IDXGRP = ADS_IGRP_TOOL_INFO_WRITE THEN (* 16#80040000  *)

		(* Tool data request from CNC *)   (* nicht bearbeiten, sondern sofort beantworten *)
		pToolId		:= Rind.DATAADDR;
		BasicToolId	:= pToolId^.basic;
		RRes.LEN			:= SIZEOF(pToolId^);
		RRes.DATAADDR	:= pToolId;
		RRes.RESULT		:= ADS_RDWRT_IND_NO_ERROR;
		bRes := TRUE;
		fbRTrigD(clk := FALSE);


	(*----- CNC tool data request with D<i>-----*)
	(* CNC fordert Werkzeuggeometriedaten aufgrund D<i> an *)
	ELSIF Rind.IDXGRP = ADS_IGRP_TOOL_DESC_READ AND
			NOT bToolData AND NOT bOldToolData THEN   (* wait until all old request are answered *)
		(* Tool data request from CNC *)
		pToolReq		:= Rind.DATAADDR;
		BasicToolId	:= pToolReq^.id.basic;
		fbRTrigD(clk := TRUE);
		IF fbRTrigD.Q THEN
			oldTool := aktTool;
			oldTool.tool_desc.param := pToolReq^.param;			(* Parameter Array aus der CNC in oldTool übernehmen *)						
			d1 := d1 + 1;
			nToolRequestID := BasicToolId;
			bToolData := TRUE;										(* start data transfer from HMI to PLC *)
		END_IF

		IF NOT bToolData THEN									(* bToolData wird false, wenn HMI Tool Daten gesendet hat (in die Struktur aktTool) *)

			RRes.LEN			:= SIZEOF(aktTool.tool_desc);
			RRes.DATAADDR	:= ADR(aktTool.tool_desc);
			RRes.RESULT		:= ADS_RDWRT_IND_NO_ERROR;
			bRes := TRUE;
			fbRTrigD(clk := FALSE);

			pos := DINT_TO_INT( aktTool.pos) ;					(* Position im Magazin *)

			
			(* Example for using additional parameters param[i] *)
			
			(*
			aktTool.tool_desc.param[4] := WkzWechslerPos1[pos * 4 ];		(* Z - AbholPos im Magazin *)
			aktTool.tool_desc.param[3] := WkzWechslerPos1[(pos * 4) - 1 ];	(* Z - AblagePos im Magazin *)
			aktTool.tool_desc.param[2] := WkzWechslerPos1[(pos * 4) - 2 ];	(* Y - Pos im Magazin *)
			aktTool.tool_desc.param[1] := WkzWechslerPos1[(pos * 4) - 3];	(* X - POS im Magazin *)
			*)
			
			(* Delta verrechnen, da in der CNC nur eine Länge ohne Delta existiert *)
			aktTool.tool_desc.laenge := aktTool.laenge + aktTool.laenge_delta;
			aktTool.tool_desc.radius := aktTool.radius + aktTool.radius_delta;

			IF aktTool.tool_desc.valid THEN
				VE_Tool 			:= DINT_TO_UINT( aktTool.tool_desc.tool_id.basic );
				nToolInCnc := aktTool.tool_desc.tool_id.basic;
				nToolInCncSister := aktTool.tool_desc.tool_id.sister;
			END_IF
		END_IF

	(*----- CNC tool life -----*)
	(* CNC aktualisiert die Werkzeugstanddaten nach Anwahl eines anderen Werkzeugs T<i> *)
	ELSIF Rind.IDXGRP = ADS_IGRP_TOOL_LIFE_DATA_WRITE THEN
		fbRTrigD(clk := FALSE);
		t1 := t1 + 1;

		(* CNC writes tool life data *)
		pToolLife := Rind.DATAADDR;
		BasicToolId := pToolLife^.tool_id.basic;
		SisterToolID := pToolLife^.tool_id.sister;

		(* no data transmitted in the response *)
		RRes.LEN			:= 0;
		RRes.DATAADDR	:= 0;

		IF BasicToolId = oldTool.tool_desc.tool_id.basic AND NOT bOldToolData THEN
			(* actualize tool life data *)
			oldTool.tool_life.dist_used := oldTool.tool_life.dist_used + pToolLife^.dist_used;
			oldTool.tool_life.time_used := oldTool.tool_life.time_used + pToolLife^.time_used;
			(* Ist das Werkzeug noch gültig ? *)
			IF oldTool.dist_max > 0 AND (oldTool.tool_life.dist_used > oldTool.dist_max) THEN
				oldTool.tool_desc.valid := FALSE;
			END_IF
			IF oldTool.time_max > 0 AND (oldTool.tool_life.time_used > oldTool.time_max) THEN
				oldTool.tool_desc.valid := FALSE;
			END_IF
			fbRTrigOldData(clk := TRUE);

			IF fbRTrigOldData.Q THEN
				bOldToolData := TRUE;
			END_IF

			RRes.RESULT := ADS_RDWRT_IND_NO_ERROR;
			IF NOT bOldToolData THEN
				bRes := TRUE;
				fbRTrigOldData(clk := FALSE);
			END_IF

		ELSE
			RRes.RESULT := WZV_TOOL_ID_BASIC_INVALID;
			fbRTrigOldData(clk := FALSE);
			bRes := TRUE;
		END_IF
	ELSE
		(* Unknown indexgroup, just send an response *)
		RRes.LEN			:= 0;
		RRes.DATAADDR	:= 0;
		RRes.RESULT		:= ADS_RDWRT_IND_UNKNOWN_INDEXGROUP;
	END_IF
END_IF


RRes(RESPOND:=bRes);

IF bRes THEN
	RRes(RESPOND:=FALSE);
	Rind(CLEAR:=TRUE);
	Rind(CLEAR:=FALSE);
END_IF

END_PROGRAM

// ---- CNC Beckhoff/1 Init/HLI3_UserInitialisation.TcPOU
FUNCTION HLI3_UserInitialisation : BOOL
VAR
	idx: UDINT;
END_VAR

(* ========================================================= *)
(*    FUN: HLI_UserInitialisation                            *)
(* --------------------------------------------------------- *)
(*   Desc:                                                   *)
(* Author: MK                                                *)
(*   Date: 18.07.2002                                        *)
(*   Rev.: 1.0 												 *)
(*         1.1 MiB 19.12.2012 Tc3 Anpassung                  *)
(*         1.2 TV 30.06.2015  Function call SetChannelControl*)
(*							  in a For Loop					 *)											  							  
(* ========================================================= *)

(* please do reset the plc program, if you change something in this module
	or in modules are in the sublevel *)

(* Axis Control *)	
HLI3_SetAxisControlToPlc();	
	
FOR idx := 0 TO gNrch - 1 DO
	HLI3_SetChannelControlToPlc(nChan:=UDINT_TO_INT(idx));
END_FOR

HLI3_UserInitialisation := TRUE;

END_FUNCTION

// ---- CNC Beckhoff/1 Init/HLI3_SetAxisControlToPlc.TcPOU
FUNCTION HLI3_SetAxisControlToPlc : BOOL
VAR
	idx: UDINT;
END_VAR

(* ========================================================= *)
(*    FUN: HLI3_SetAxisControlToPlc                          *)
(* --------------------------------------------------------- *)
(*   Desc:                                                   *)
(*   Author: MiB                                             *)
(*   Date: 19.11.2012                                        *)
(*   Rev.: 1.0                                               *)
(* ========================================================= *)

(* control to the plc *)
FOR idx := 0 TO gNrAx - 1 DO

	IF (idx < INT_TO_UDINT(HLI_SYS_AX_MAX)) THEN 
		IF gpAx[idx] <> 0 THEN						// check for zero pointer
			// PLC_Present for all axis
			gpAx[idx]^.head.plc_present_w 								:= TRUE;
		
			(* declare axis for reference *)
			gpAx[idx]^.lr_mc_control.reference_cam.enable_w 			:= TRUE;
	
			(* enable signals for real drives *)
			gpAx[idx]^.lr_mc_control.torque_permission.enable_w			:= TRUE;
			gpAx[idx]^.lr_mc_control.release_feedhold.enable_w 			:= TRUE;
			gpAx[idx]^.lr_mc_control.drive_on.enable_w 					:= TRUE;
			
			(* set reference postion offset *)
			gpAx[idx]^.lr_mc_control.set_reference_position.enable_w	:= TRUE;
			gpAx[idx]^.lr_mc_control.refpos_position.enable_w			:= TRUE;
			gpAx[idx]^.lr_mc_control.reference_cam.enable_w				:= TRUE;
			
			(* enable external commanding of an axis *)
			gpAx[idx]^.lr_mc_control.add_cmd_values.enable_w 			:= TRUE;
	
			(* enable the axis to tracking operation (follow up) *)
			gpAx[idx]^.lr_mc_control.follow_up.enable_w 				:= TRUE;
		END_IF
	END_IF
END_FOR

HLI3_SetAxisControlToPlc												:= TRUE;

END_FUNCTION

// ---- CNC Beckhoff/1 Init/HLI3_SetChannelControlToPlc.TcPOU
FUNCTION HLI3_SetChannelControlToPlc : BOOL
VAR_INPUT
	nChan: INT;
END_VAR

(* ========================================================= *)
(*    FUN: HLI3_SetChannelControlToPlc                       *)
(* --------------------------------------------------------- *)
(*   Desc:                                                   *)
(* Author: MK                                                *)
(*   Date: 18.07.2002                                        *)
(*   Rev.: 1.0                                               *)
(*   Date: 19.11.2012                                        *)
(*   Rev.: 1.1 MiB TC3 0 based index                         *)
(* ========================================================= *)


IF (NOT HLI3_CheckChannelValid(nChannel := nCHan)) THEN
	HLI3_SetChannelControlToPlc											:= FALSE;
	RETURN; (* A b b r u c h *)
END_IF


(* PLC_Present for the channel *)
gpCh[nChan]^.head.plc_present_w 									:= TRUE;

(* reset *)
gpCh[nChan]^.bahn_lc_control.plc_reset.enable_w 					:= TRUE;
gpCh[nChan]^.channel_mc_control.mode_and_state.enable_w				:= TRUE;

(* override *)
gpCh[nChan]^.bahn_mc_control.override_feedrate.enable_w 			:= TRUE;

(* FeedHold *)
gpCh[nChan]^.bahn_mc_control.feedhold.enable_w 					:= TRUE;

(* Single Step *)
gpCh[nChan]^.bahn_mc_control.single_block.enable_w 				:= TRUE;

(* BackwardMotion *)
gpCh[nChan]^.bahn_mc_control.backward_motion.enable_w 			:= TRUE;

(* ReducedFeed *)
gpCh[nChan]^.bahn_mc_control.reduced_speed.enable_w 				:= TRUE;

(* Handwheel *)
gpCh[nChan]^.hb_mc_control.handwheel_incs[0].enable_w 			:= TRUE;

(* Channel switch "jog of path" *)
gpCh[nChan]^.bahn_mc_control.suspend_axis_output.enable_w 		:= TRUE;

(* logon for error messages *)
gpCh[nChan]^.mc_error.enable_w 									:= TRUE;

(* program block ignore *)
gpCh[nChan]^.decoder_mc_control.program_block_ignore.enable_w	:= TRUE;

(* Syntax Check *)
gpCh[nChan]^.decoder_mc_control.execution_mode.enable_w			:= TRUE;

(* Optional stop M01 *)
gpCh[nChan]^.bahn_mc_control.m01_stop_enable.enable_w			:= TRUE;

(* Emergency Stop *)
gpCh[nChan]^.bahn_mc_control.emergency_stop.enable_w				:= TRUE;

HLI3_SetChannelControlToPlc 												:= TRUE;

END_FUNCTION

// ---- CNC Beckhoff/9 Mis/ADSLOG.TcPOU
FUNCTION ADSLOG : BOOL
VAR_INPUT
	strMsg: STRING;
	nDINT: DINT;
	strArg: STRING;
END_VAR

RETURN;

IF strArg = '' THEN
	ADSLOGDINT( msgCtrlMask :=    ADSLOG_MSGTYPE_MSGBOX
	                           OR ADSLOG_MSGTYPE_LOG,
				msgFmtStr   := strMsg,
				dintArg     := nDINT);
ELSE
	ADSLOGSTR( msgCtrlMask :=    ADSLOG_MSGTYPE_MSGBOX
	                          OR ADSLOG_MSGTYPE_LOG,
				msgFmtStr := strMsg,
				strArg := strArg);
END_IF

END_FUNCTION

// ---- CNC Beckhoff/9 Mis/HLI3_CheckAxisValid.TcPOU
FUNCTION HLI3_CheckAxisValid : BOOL
VAR_INPUT
	nHliAxisIdx: INT;
END_VAR

(* ========================================================= *)
(*    FUN: HLI3_CheckAxisValid                               *)
(* --------------------------------------------------------- *)
(*   Desc: Check if axis ID is valid for HLI access       	 *)
(*   Author: MiB                                             *)
(*   Date: 19.11.2012                                        *)
(*   Rev.: 1.0                                               *)
(* --------------------------------------------------------- *)
(*   Desc: Corrected IF statement (line 17)		 	      	 *)
(*   Author: RCH                                             *)
(*   Date: 16.09.2013                                        *)
(*   Rev.: 1.1                                               *)
(* ========================================================= *)
IF (nHliAxisIdx < 0) OR 
	(nHliAxisIdx >= UDINT_TO_INT(gNrAx) ) OR		(* check for axis no *)
    (gpAx[nHliAxisIdx] = 0) 				  (* check for zero pointer *)
THEN
	HLI3_CheckAxisValid:= FALSE;
	RETURN; (* A b b r u c h *)
ELSE
	HLI3_CheckAxisValid := TRUE;
	RETURN;
END_IF

END_FUNCTION

// ---- CNC Beckhoff/PRG_AxesHandler.TcPOU
PROGRAM PRG_AxesHandler
VAR
	nHliAxisIdx					: INT;		
	fbSetAxisRelease			: ARRAY[0..HLI_SYS_AX_MAXIDX] OF HLI3_SetAxisRelease;
	
	nFirstSpindle				: INT := -1;
	fbHandleSpindleTechno		: HLI3_HandleSpindleTechnoGearChange;
	M3,M4,M5,M19				: BOOL;
	MDummy						: BOOL;
	M40, M41, M42, M43, M44, M45: BOOL;
	(*
	fbHandleSpindleTechnoPlcSp	: HLI3_HandleSpindleTechno;
	SM3,SM4,SM5,SM19			: bool; 
	*)
END_VAR

(****************************************************************************************)
(* POU:		PRG_AxesHandler                     										*)
(* Type:	PRG																			*)
(* Author: 	TV,MiB                                             							*)
(* Date: 	03.02.14																	*)
(* Rev.: 	1.1                                               							*)
(* ------------------------------------------------------------------------------------ *)
(* Desc:	Description																	*)
(****************************************************************************************)

(****************************************************************************************)
(*							Release of all reachable axes								*)
(****************************************************************************************)
FOR nHliAxisIdx := 0 TO HLI_SYS_AX_MAXIDX DO
	fbSetAxisRelease[nHliAxisIdx](
		bEnable:= PLCAxisEnable, 
		nHliAxisIdx:= nHliAxisIdx);	
		IF HLI3_CheckAxisValid(nHliAxisIdx) THEN
			IF nFirstSpindle = -1 AND gpAx[nHliAxisIdx]^.ipo_state.spindle_axis_r THEN  (* store HLIIndex of first spindle *)
				nFirstSpindle := nHliAxisIdx;
			END_IF
		END_IF
END_FOR



(* if there exits spindles use the first one for spindleoverride *)
IF nFirstSpindle <> -1 THEN
	HLI3_SetAxisOverride(nHliAxisIdx:= nFirstSpindle , nOverride:= PLCSpindleOverride *10);

	fbHandleSpindleTechno(
		nHliAxisIdx:=nFirstSpindle , 		
		bIsChannelSpecific:= FALSE, 
		nRevolution=> , 
		nPosition=> , 
		bError=> , 
		nErrorId=> , 
		M03:= M3, 
		M04:= M4, 
		M05:= M5, 
		M19:= M19,
		M40 := M40,
		M41 := M41,
		M42 := M42,
		M43 := M43,
		M44 := M44,
		M45 := M45,
		); 
	(* acknowledge all spindle M funnctions immediately *)
	M3 := FALSE;  
	M4 := FALSE;
	M5 := FALSE;
	M19 := FALSE;
END_IF



(* Howto use plc controlled spindle : *)
(*
fbHandleSpindleTechnoPlcSp(
	nHliAxisIdx:= 0 , 
	nHliChannelIdx:= 0 , 
	bIsChannelSpecific:= TRUE, 
	nLogAxisNoChannelSpecific:= 95 , 
	bHandleGearChange:= FALSE , 
	bChannelReset:= FALSE, 
	nRevolution=> , 
	nPosition=> , 
	bError=> , 
	nErrorId=> , 
	M03:= SM3, 
	M04:= SM4, 
	M05:= SM5, 
	M19:= SM19);
*)

END_PROGRAM

// ---- CNC Beckhoff/3 Control/HLI3_SetAxisRelease.TcPOU
FUNCTION_BLOCK HLI3_SetAxisRelease
VAR_INPUT
	bEnable: BOOL;
	nHliAxisIdx: INT;
END_VAR
VAR_OUTPUT
	bAxisIsReady: BOOL;
	bAxisIsEnabled: BOOL;
	bAxisHasError: BOOL;
	nDriveType: UDINT;
	bError: BOOL;
	nErrorId: UDINT;
	nErrorState: UINT;
END_VAR
VAR
	bReadyForPowerOn: BOOL;
	bReadyForControlLoopOn: BOOL;
	nHliAxisIdxOld: INT;
	nState: UINT;
	nStateOld: UINT;
	tActiveTimeOut: TIME := TIME#5s0ms;
	wDriveState: WORD;
	fbTonTimeOut: TON;
END_VAR
VAR CONSTANT
	ERR_INVALID_AXIS_IDX: UDINT := 10000;
	ERR_UNSUPPORTED_DRIVE: UDINT := 10001;
	ERR_TIME_OUT: UDINT := 10002;
END_VAR

(****************************************************************************************)
(* POU:		HLI3_SetAxisRelease                      									*)
(* Type:	Function block																*)
(* Author: 	HR																			*)
(* Date: 	14/01/10																	*)
(* Rev.: 	1.0																			*)
(* ------------------------------------------------------------------------------------ *)
(* Author: 	TV																			*)
(* Date: 	14/04/11																	*)
(* Rev.: 	1.1																			*)
(* 			Implementation for terminal drives											*)
(* ------------------------------------------------------------------------------------ *)
(* Author: 	HR																			*)
(* Date: 	14/08/27																	*)
(* Rev.: 	1.2																			*)
(* 			Fixed terminal drive issue --> According to the ISG docs terminal drives	*)
(*			are supported by means of the torque permission control unit only! There-	*)
(*			fore this has to be switched by the 'bEnable' input. Tested with EL7041		*)
(* ------------------------------------------------------------------------------------ *)
(* Author: 	MiB																			*)
(* Date: 	16/04/06																	*)
(* Rev.: 	1.2																			*)
(* 			Enable follow up only for non simulation axis								*)
(* ------------------------------------------------------------------------------------ *)		
(* Desc:	Sets axes release and follow up mode using the axis specific control units 	*)
(*			'.lr_mc_control.torque_permission', 'lr_mc_control.release_feedhold',		*)
(*			'lr_mc_control.drive_on' and 'lr_mc_control.follow_up' depending on the 	*)
(*			subsequent drive type (e.g. Sercos,...). The following drive type are 		*)
(*			supported:																	*)
(*				+ Sercos and SoE														*)
(*				+ CanOpen and CoE (according to CiA402 drive profile)					*)
(*				+ Simulation drives														*)
(*																						*)
(*			This function block may raise the following error numbers					*)
(*				+ 10000	--> Invalid 'nHliAxisIdx'										*)
(*				+ 10001 --> Unsupported drive type										*)
(*				+ 10002 --> Time out while setting axis release							*)
(*																						*)
(*			IMPORTANT: This function block does not implement any state specific en- or	*)
(*			disabling of the drive. It simply tries to enable the subsequent axis as	*)
(*			long as input variable 'bEnable' is TRUE. That means it won´t disable the 	*)
(*			drive in case of any errors or loss prerequisited operation conditions (e.g.*)
(*			power supply). It is assumed that the drive will handle those situations	*)
(*			internally!																	*)
(*				  																		*)
(* 			Tested with following drives:												*)
(*																						*)
(*			VENDOR				MAKE					FW-VERSION			COM-SYS 	*)
(* 			------				----					----------			-------		*)
(* 			Beckhoff			AX5xxx					2.03 (B26)			SoE			*)
(* 			Beckhoff			EL7201					03					CoE			*)
(*			Beckhoff			EL7041					10					Terminal	*)	
(* 			ELMO				Gold					01.01.07.12			CoE			*)
(****************************************************************************************)

(****************************************************************************************)
(*									Check axis index									*)
(****************************************************************************************)
IF NOT HLI3_CheckAxisValid(nHliAxisIdx) THEN
	bError		:= TRUE;
	nErrorId	:= ERR_INVALID_AXIS_IDX;
	RETURN;
END_IF

(****************************************************************************************)
(*										Clear errors									*)
(****************************************************************************************)
IF bError THEN
	CASE nErrorId OF
	 (* -------------------------------------------------------------------------------	*)
	 ERR_INVALID_AXIS_IDX:
	 	(* Reset invalid HLI axis index error as soon as this line has been hit!		*)
		AC_ClearError();
		
	(* -------------------------------------------------------------------------------	*)
	 ERR_UNSUPPORTED_DRIVE:
		(* Reset unsupported drive type error in case the HLI axis index has been 		*)
		(* changed!																		*)
		IF (nHliAxisIdx <> nHliAxisIdxOld) THEN
			nHliAxisIdxOld	:= nHliAxisIdx;
			AC_ClearError();
		END_IF
 
	(* -------------------------------------------------------------------------------	*) 
	 ERR_TIME_OUT:
 		(* Will be resetted individually by each drive type specific action!			*)
	END_CASE
END_IF

(****************************************************************************************)
(*								Switch follow up mode 									*)
(****************************************************************************************)
IF gpAx[nHliAxisIdx]^.lr_state.drive_type_r = 4 THEN   (* type == 4 -> simulation axis -> don't enable follow up mode *)
	gpAx[nHliAxisIdx]^.lr_mc_control.follow_up.command_w := FALSE;
ELSE
	gpAx[nHliAxisIdx]^.lr_mc_control.follow_up.command_w := NOT bEnable;
END_IF

(****************************************************************************************)
(*						Copy axis state information to local variables					*)
(****************************************************************************************)
wDriveState				:= gpAx[nHliAxisIdx]^.lr_state.native_drive_state_r;
nDriveType				:= gpAx[nHliAxisIdx]^.lr_state.drive_type_r;
bAxisHasError			:= gpAx[nHliAxisIdx]^.lr_state.error_r;
bReadyForPowerOn		:= gpAx[nHliAxisIdx]^.lr_state.ready_for_power_on_r;
bReadyForControlLoopOn	:= gpAx[nHliAxisIdx]^.lr_state.ready_for_control_loop_on_r;

(****************************************************************************************)
(*							 Constant timeout implementation							*)
(****************************************************************************************)
IF (nStateOld <> nState) THEN
	nStateOld	:= nState;
	fbTonTimeOut(IN := FALSE);
END_IF

fbTonTimeOut
	(IN := TRUE,
	 PT := tActiveTimeOut
	);

(****************************************************************************************)
(*								Drive type specific axis release						*)
(****************************************************************************************)
CASE nDriveType OF
	HLI_DRIVE_CANOPEN	: AC_CanOpenDrive();
	HLI_DRIVE_SERCOS	: AC_SercosDrive();
	HLI_DRIVE_SIMU		: AC_SercosDrive();
	HLI_DRIVE_TERMINAL  : AC_TerminalDrive();
ELSE
	bError				:= TRUE;
	nErrorId			:= ERR_UNSUPPORTED_DRIVE;
END_CASE

ACTION AC_TerminalDrive:
(****************************************************************************************)
(*										Status data										*)
(****************************************************************************************)
(* Since there is no feedback available on the HLI axis enabled state wiöö be emulated!	*)
bAxisIsEnabled	:= bEnable;
bAxisIsReady	:= FALSE;
 
(****************************************************************************************)
(*										Command data									*)
(****************************************************************************************)
(* Terminal drives are supported by the torque permission control unit only!			*)
gpAx[nHliAxisIdx]^.lr_mc_control.torque_permission.command_w	:= bEnable;
gpAx[nHliAxisIdx]^.lr_mc_control.release_feedhold.command_w		:= FALSE;
gpAx[nHliAxisIdx]^.lr_mc_control.drive_on.command_w				:= FALSE;
END_ACTION

ACTION AC_ClearError:
THIS^.bError		:= FALSE;
THIS^.nErrorId		:= 0;
THIS^.nErrorState	:= 0;
END_ACTION

ACTION AC_CanOpenDrive:
(****************************************************************************************)
(*										Status data										*)
(****************************************************************************************)
(* Ready state is signalled if the drive´s state is unequal to 'Not ready to switch on'	*)
bAxisIsReady	:= bReadyForControlLoopOn; 
 
(* Enabled state is derived from state 'Operation enabled' (information provided via	*)
(* HLI) and from status word bit no. 01 (switched on)!									*)
bAxisIsEnabled	:= bReadyForControlLoopOn AND bReadyForPowerOn AND wDriveState.1;

(****************************************************************************************)
(*						Command data (CanOpen requires a state machine)					*)
(****************************************************************************************)
(* Switch back to initial state in case the user want´s to disable the drive or an axis	*)
(* error occured, which requires a new srun of the sequence!							*)
IF NOT bEnable OR wDriveState.3 THEN
	nState				:= 0;
END_IF

CASE nState OF
 (* -----------------------------------------------------------------------------------	*)
 0: (* INIT *)
 	gpAx[nHliAxisIdx]^.lr_mc_control.torque_permission.command_w	:= FALSE;
 	gpAx[nHliAxisIdx]^.lr_mc_control.release_feedhold.command_w		:= FALSE;
	
	(* Start sequence in case the user wants to enable the drive and there is no error.	*)
 	IF bEnable AND NOT wDriveState.3 AND bAxisIsReady THEN
		(* Set time out once! *)
		tActiveTimeOut	:= T#2S;	
	
		// Switch on disabled???
		IF wDriveState.6 THEN
			nState		:= 10;
		//Ready to switch on???
		ELSIF wDriveState.0 THEN
			nState		:= 20;
		//Switched on???
		ELSIF wDriveState.1 THEN
			nState		:= 30;
		//Operation enabled???
		ELSIF wDriveState.2 THEN
			nState		:= 40;
		END_IF
	END_IF
	
 (* -----------------------------------------------------------------------------------	*)
 10: (* DRIVE IN 'Switch on disabled' STATE *)
 	gpAx[nHliAxisIdx]^.lr_mc_control.drive_on.command_w				:= TRUE;
 
	IF wDriveState.0 THEN
		nState			:= 20; 
	ELSIF fbTonTimeOut.Q THEN
		bError			:= TRUE;
		nErrorId		:= ERR_TIME_OUT;
		nErrorState		:= nState;
		nState			:= 0;
	END_IF
	
(* -----------------------------------------------------------------------------------	*)
 20: (* DRIVE IN 'Ready to switch on' STATE *)
 	gpAx[nHliAxisIdx]^.lr_mc_control.torque_permission.command_w	:= TRUE;
	
	IF wDriveState.1 THEN
		nState			:= 30; 
	ELSIF fbTonTimeOut.Q THEN
		bError			:= TRUE;
		nErrorId		:= ERR_TIME_OUT;
		nErrorState		:= nState;
		nState			:= 0;
	END_IF
	
 (* -----------------------------------------------------------------------------------	*)
 30: (* DRIVE IN 'Switched on' STATE *)
 	gpAx[nHliAxisIdx]^.lr_mc_control.release_feedhold.command_w		:= TRUE;
	
	IF wDriveState.2 THEN
		nState			:= 40; 
	ELSIF fbTonTimeOut.Q THEN
		bError			:= TRUE;
		nErrorId		:= ERR_TIME_OUT;
		nErrorState		:= nState;
		nState			:= 0;
	END_IF
	
 (* -----------------------------------------------------------------------------------	*)
 40: (* DRIVE IN 'Operation enabled' STATE *)
	AC_ClearError();
	
END_CASE
END_ACTION

ACTION AC_SercosDrive:
(****************************************************************************************)
(*										Status data										*)
(****************************************************************************************)
(* Ready state is derived from status word bit 15!										*)
bAxisIsReady	:= bReadyForControlLoopOn; 
 
(* Enabled state is derived from status word bits 14 and 15. IMPORTANT: In order to 	*)
(* take status word bit 03 into account  - which represents the time needed for 		*)
(* releasing the brake - axis specific parameter 'antr.sercos.evaluate_drive_follows_	*)
(* cmd' has to be set!!!																*) 
bAxisIsEnabled	:= bReadyForControlLoopOn AND bReadyForPowerOn;
 
(****************************************************************************************)
(*										Command data									*)
(****************************************************************************************)
(* ControlBit no. 14 is set statically in order to provide torque supported stopping of	*)
(* in case someone disables the axis during movement!									*) 
gpAx[nHliAxisIdx]^.lr_mc_control.torque_permission.command_w	:= TRUE;

(* Only control bits 13 and 15 are being (re-)set in order to achieve axis enabling!	*)
gpAx[nHliAxisIdx]^.lr_mc_control.release_feedhold.command_w		:= bEnable;
gpAx[nHliAxisIdx]^.lr_mc_control.drive_on.command_w				:= bEnable;
END_ACTION

END_FUNCTION_BLOCK

// ---- CNC Beckhoff/3 Control/HLI3_HandleSpindleTechnoGearchange.TcPOU
FUNCTION_BLOCK HLI3_HandleSpindleTechnoGearchange EXTENDS HLI3_HandleSpindleTechno
VAR_INPUT
END_VAR
VAR_OUTPUT
END_VAR
VAR_IN_OUT
		/// Raises if the cnc program encounters a M40 for the relevant spindle. Reset this for acknowledge 
	M40: BOOL;
	/// Raises if the cnc program encounters a M41 for the relevant spindle. Reset this for acknowledge 
	M41: BOOL;
	/// Raises if the cnc program encounters a M42 for the relevant spindle. Reset this for acknowledge 
	M42: BOOL;
	/// Raises if the cnc program encounters a M43 for the relevant spindle. Reset this for acknowledge 
	M43: BOOL;
	/// Raises if the cnc program encounters a M44 for the relevant spindle. Reset this for acknowledge 
	M44: BOOL;
	/// Raises if the cnc program encounters a M45 for the relevant spindle. Reset this for acknowledge 
	M45: BOOL;	
END_VAR
VAR
END_VAR

(* Date:	15/03/05																	*)
(* Author:	MiB																			*)
(* Rev:		1.0																			*)
(* ------------------------------------------------------------------------------------ *)
(* Desc 	Handling of spindle gear change M functions M40 - M45.						*)
(*			extends HLI3_SpindleTechno													*)
(*			overwrites the internal pointers to M40..M45 to VAR_IN_OUT					*)


SUPER^.pM40 := ADR(M40);
SUPER^.pM41 := ADR(M41);
SUPER^.pM42 := ADR(M42);
SUPER^.pM43 := ADR(M43);
SUPER^.pM44 := ADR(M44);
SUPER^.pM45 := ADR(M45);

A_HandleTechno();

END_FUNCTION_BLOCK

// ---- CNC Beckhoff/3 Control/HLI3_HandleSpindleTechno.TcPOU
FUNCTION_BLOCK HLI3_HandleSpindleTechno
VAR_INPUT
	/// Logical axis number of the plc spindle 
	nHliAxisIdx: INT;
	/// The channel which commands the spindle, only used if 'bIsChannelSpecific' set TRUE 
	nHliChannelIdx: INT;
	/// Has to be set TRUE if the spindel intechno function is transmitted via the channel specific section of the HLI
	bIsChannelSpecific: BOOL;
	/// if using a plc controlled spindle: configured log_ax_nr in channel list 
	nLogAxisNoChannelSpecific: INT;
	/// Has to be set TRUE if zthis FB should car about gear change M functions M40 - M45
	bHandleGearChange: BOOL;
	/// Resets all internal states and variables of this function block 
	bChannelReset: BOOL;
END_VAR
VAR_OUTPUT
	/// Returns the commanded revolution programmed with a M03 or M05 [] 
	nRevolution: DINT;
	/// Returns the target position programmed with a M19 [0.1µm] or [] 
	nPosition: DINT;
	/// Error flag 
	bError: BOOL;
	/// Error id 
	nErrorId: UDINT;
END_VAR
VAR_IN_OUT
	/// Raises if the cnc program encounters a M03 for the relevant spindle. Reset this for acknowledge 
	M03: BOOL;
	/// Raises if the cnc program encounters a M04 for the relevant spindle. Reset this for acknowledge 
	M04: BOOL;
	/// Raises if the cnc program encounters a M05 for the relevant spindle. Reset this for acknowledge 
	M05: BOOL;
	/// Raises if the cnc program encounters a M19 for the relevant spindle. Reset this for acknowledge 
	M19: BOOL;
END_VAR
VAR
	/// Raises if the cnc program encounters a M40 for the relevant spindle. Reset this for acknowledge 
	pM40: POINTER TO BOOL;
	/// Raises if the cnc program encounters a M41 for the relevant spindle. Reset this for acknowledge 
	pM41: POINTER TO BOOL;
	/// Raises if the cnc program encounters a M42 for the relevant spindle. Reset this for acknowledge 
	pM42: POINTER TO BOOL;
	/// Raises if the cnc program encounters a M43 for the relevant spindle. Reset this for acknowledge 
	pM43: POINTER TO BOOL;
	/// Raises if the cnc program encounters a M44 for the relevant spindle. Reset this for acknowledge 
	pM44: POINTER TO BOOL;
	/// Raises if the cnc program encounters a M45 for the relevant spindle. Reset this for acknowledge 
	pM45: POINTER TO BOOL;	


	/// Number of open technology functions 
	nOpenTechnoCount: UINT;
	/// Internal acknowledge signal 
	bAcknowledge: BOOL;
	/// Internal state of M03 request 
	M03_Internal: BOOL;
	/// Internal state of M04 request 
	M04_Internal: BOOL;
	/// Internal state of M05 request 
	M05_Internal: BOOL;
	/// Internal state of M19 request 
	M19_Internal: BOOL;
	/// Internal state of M19 request 
	M40_Internal: BOOL;
	/// Internal state of M19 request 
	M41_Internal: BOOL;
	/// Internal state of M19 request 
	M42_Internal: BOOL;
	/// Internal state of M19 request 
	M43_Internal: BOOL;
	/// Internal state of M19 request 
	M44_Internal: BOOL;
	/// Internal state of M19 request 
	M45_Internal: BOOL;
	/// Index of axis specific HLI area 
	nHliAxIfcIdx: UDINT;
	/// Index of axis specific technology function at HLI 
	nTechFctMaxIdx: UINT;
	/// Counting variable for loop processing 
	nLoop: UINT;
	/// Pointer to technology function data 
	pActTechnoUnit: POINTER TO TECHNO_UNIT_AX;
	/// Pointer to spindle specific data 
	pSProcess: POINTER TO HLI_S_PROZESS;
	pMProcess: POINTER TO HLI_M_H_PROZESS;
	/// Rising trigger of input 'bChannelReset' 
	fbRtrigChannelReset: R_TRIG;
	
	bFirstRun : BOOL := TRUE;
	dummyM40: BOOL;
	dummyM41: BOOL;
	dummyM42: BOOL;
	dummyM43: BOOL;
	dummyM44: BOOL;
	dummyM45: BOOL;
	
END_VAR

(****************************************************************************************)
(* POU:		HLI3_HandlePlcSpindle                      									*)
(* Type:	Function Block																*)
(* Author: 	HR, MiB, TV																    *)
(* Date: 	10/11/10																	*)
(* Rev.: 	1.0																			*)
(* Rev.: 	1.6	14/10/23    															*)
(* ------------------------------------------------------------------------------------ *)
(* Desc:	Function block for handling technology functions of PLC spindles. It works	*)
(*			properly if there is a ation axis in the configuration. The logical 		*)
(*			axis no. 'n' of that axis is used to indetify that spindle in this function	*)
(*			block. This implies a spindle configuration like the folowing:				*)
(*				spdl_anzahl                         1	(maybe more?)					*)
(*				main_spindle_ax_nr                  n	(enter right value there)		*)
(*				main_spindle_name                   S									*)
(*				spindle_m_fct_free                  0									*)
(*				spindel[0].bezeichnung              S1									*)
(*				spindel[0].log_achs_nr              n	(enter right value there)		*)
(*				spindel[0].plc_control              1									*)
(*																						*)
(*			The function block may raise some errors specified by an error id:			*)
(*				+ 10000: axis number not valid!											*)
(*																						*)
(****************************************************************************************)
(* Date:	13/09/16																	*)
(* Author:	RCH																			*)
(* Rev:		1.1																			*)
(* ------------------------------------------------------------------------------------ *)
(* Desc 	Renamed, according to Tc2 version. This FB also works for CNC spindles with	*) 
(*			S or M functions set to inform PLC. 										*)
(****************************************************************************************)
(* Date:	13/09/16																	*)
(* Author:	RCH																			*)
(* Rev:		1.2																			*)
(* ------------------------------------------------------------------------------------ *)
(* Desc 	Introduced new input parameters 'bIsChannelSpecific' and 'nChannelNo' in 	*)
(*			order to make this FB work for PLC spindles which are sending synch.		*)
(*			requests via the channel specific section of the HLI. Here the spindle		*)
(* 			specific parameters have to be set as follows:								*)
(*				spindel[n].plc_control            1			(P-CHAN-00069)				*)
(*				spindel[n].log_achs_nr            m			(P-CHAN-00036)				*)
(*																						*)
(*			The logical axis number in P-CHAN-00036 used for such a spindle must not be	*)
(*			lower than one and must not be used by any other axis. This FB works if the	*)
(*			value of this logical axis number fits the parameter 'nHliAxisIdx' only!	*)
(* 																						*)
(*			In order to guarantee save HLI access the following new error codes have	*)
(*			been introduced:															*)
(*				+ 20000: Channel no lower than one!										*)
(*				+ 20001: Channel number exceeds number of configured channels.			*)
(*				+ 20002: No HLI data for channel.										*)
(****************************************************************************************)
(* Date:	14/01/22																	*)
(* Author:	TV																			*)
(* Rev:		1.3																			*)
(* ------------------------------------------------------------------------------------ *)
(* Desc:	bugfix in function to check nHLIAxisIdx and LogAxisId						*) 
(****************************************************************************************)
(* Date:	14/09/10																	*)
(* Author:	RCH																			*)
(* Rev:		1.4																			*)
(* ------------------------------------------------------------------------------------ *)
(* Desc 	Added optional handling of spindle gear change M functions M40 - M45.		*)
(****************************************************************************************)
(* Date:	14/09/12																	*)
(* Author:	RCH																			*)
(* Rev:		1.5																			*)
(* ------------------------------------------------------------------------------------ *)
(* Desc 	Fixed bug with spindle M functions send by the channel spec. section of the	*)
(*			HLI. So far the channel specific section was used for determining the value *)
(*			of  'nTechFctMaxidx'.														*)
(****************************************************************************************)
(* Date:	14/10/23																	*)
(* Author:	MiB																			*)
(* Rev:		1.6																			*)
(* ------------------------------------------------------------------------------------ *)
(* Desc 	Introduced parameter "nLogAxisNoChannelSpecific" which allows to use a plc  *)
(*			spindle without a simulation axis for the spindle. 				 			*)
(*			This paramater is only used if "bIsChannelSpecific == true"					*)
(*																						*)
(*				spindel[n].plc_control            1			(P-CHAN-00069)				*)
(*				spindel[n].log_achs_nr            m			(P-CHAN-00036)				*)
(*																						*)
(*			The logical axis number in P-CHAN-00036 used for such a spindle must not be	*)
(*			lower than one and must not be used by any other axis. This FB works if the	*)
(*			value of this logical axis number fits the parameter 						*)
(*			'nLogAxisNoChannelSpecific' only!											*)
(****************************************************************************************)
(* Date:	15/03/05																	*)
(* Author:	MiB																			*)
(* Rev:		1.7																			*)
(* ------------------------------------------------------------------------------------ *)
(* Desc 	Removed gearchange m functions from var_in_out							    *)
(*			Created new FB HLI3_SpindleTechnoGearchange									*)
(****************************************************************************************)

(****************************************************************************************)
(*								Init Pointer to pM40..pM45								*)
(****************************************************************************************)
IF bFirstRun THEN
	bFirstRun := FALSE;
	pM40 := ADR(dummyM40);
	pM41 := ADR(dummyM41);
	pM42 := ADR(dummyM42);
	pM43 := ADR(dummyM43);
	pM44 := ADR(dummyM44);
	pM45 := ADR(dummyM45);	
END_IF

A_HandleTechno();

ACTION A_HandleTechno:

(****************************************************************************************)
(*								Cyclic reset of  error flag 							*)
(****************************************************************************************)
bError										:= FALSE;
nErrorId									:= 0;

